LIN {X 0,Y 474.616,Z 278.985,A -85,B 0,C 180,E1 -7437.787,E2 -7437.787} C_VEL
LIN {X 0,Y 474.604,Z 278.989,A -85,B 0,C 180,E1 -7440.884,E2 -7440.884} C_VEL
LIN {X 0,Y 474.635,Z 278.982,A -85,B 0,C 180,E1 -7443.627,E2 -7443.627} C_VEL
LIN {X 0,Y 474.616,Z 278.99,A -85,B 0,C 180,E1 -7446.641,E2 -7446.641} C_VEL
LIN {X 0,Y 474.636,Z 278.981,A -85,B 0,C 180,E1 -7450.089,E2 -7450.089} C_VEL
LIN {X 0,Y 474.637,Z 278.985,A -85,B 0,C 180,E1 -7451.617,E2 -7451.617} C_VEL
LIN {X 0,Y 473.97,Z 279.072,A -85,B 0,C 180,E1 -7452.326,E2 -7452.326} C_VEL
LIN {X 0,Y 471.122,Z 279.425,A -85,B 0,C 180,E1 -7453.477,E2 -7453.477} C_VEL
LIN {X 0,Y 468.71,Z 279.726,A -85,B 0,C 180,E1 -7454.406,E2 -7454.406} C_VEL
LIN {X 0,Y 467.667,Z 279.855,A -85,B 0,C 180,E1 -7455.123,E2 -7455.123} C_VEL
LIN {X 0,Y 467.579,Z 279.864,A -85,B 0,C 180,E1 -7455.365,E2 -7455.365} C_VEL
LIN {X 0,Y 467.665,Z 279.853,A -85,B 0,C 180,E1 -7457.855,E2 -7457.855} C_VEL
LIN {X 0,Y 467.663,Z 279.853,A -85,B 0,C 180,E1 -7461.357,E2 -7461.357} C_VEL
LIN {X 0,Y 467.715,Z 279.848,A -85,B 0,C 180,E1 -7463.962,E2 -7463.962} C_VEL
LIN {X 0,Y 467.84,Z 279.834,A -85,B 0,C 180,E1 -7467.417,E2 -7467.417} C_VEL
LIN {X 0,Y 467.861,Z 279.836,A -85,B 0,C 180,E1 -7470,E2 -7470} C_VEL
LIN {X 0,Y 467.838,Z 279.841,A -85,B 0,C 180,E1 -7472.583,E2 -7472.583} C_VEL
LIN {X 0,Y 467.733,Z 280.061,A -85,B 0,C 180,E1 -7473.068,E2 -7473.068} C_VEL
LIN {X 0,Y 470.913,Z 294.475,A -85,B 0,C 180,E1 -7475.781,E2 -7475.781} C_VEL
LIN {X 0,Y 471.168,Z 295.669,A -85,B 0,C 180,E1 -7475.953,E2 -7475.953} C_VEL
LIN {X 0,Y 475.313,Z 312.707,A -85,B 0,C 180,E1 -7476.456,E2 -7476.456} C_VEL
LIN {X 0,Y 476.029,Z 316.068,A -85,B 0,C 180,E1 -7476.548,E2 -7476.548} C_VEL
LIN {X 0,Y 474.23,Z 459.892,A -85,B 0,C 180,E1 -7478.817,E2 -7478.817} C_VEL
LIN {X 0,Y 473.781,Z 475.482,A -85,B 0,C 180,E1 -7479.229,E2 -7479.229} C_VEL
LIN {X 0,Y 473.147,Z 491.137,A -85,B 0,C 180,E1 -7479.835,E2 -7479.835} C_VEL
LIN {X 0,Y 472.45,Z 505.523,A -85,B 0,C 180,E1 -7480.579,E2 -7480.579} C_VEL
LIN {X 0,Y 471.64,Z 519.544,A -85,B 0,C 180,E1 -7481.496,E2 -7481.496} C_VEL
LIN {X 0,Y 470.763,Z 533.282,A -85,B 0,C 180,E1 -7482.611,E2 -7482.611} C_VEL
LIN {X 0,Y 469.923,Z 545.755,A -85,B 0,C 180,E1 -7483.844,E2 -7483.844} C_VEL
LIN {X 0,Y 469.124,Z 557.142,A -85,B 0,C 180,E1 -7485.198,E2 -7485.198} C_VEL
LIN {X 0,Y 468.452,Z 566.781,A -85,B 0,C 180,E1 -7486.561,E2 -7486.561} C_VEL
LIN {X 0,Y 467.84,Z 576.198,A -85,B 0,C 180,E1 -7488.162,E2 -7488.162} C_VEL
LIN {X 0,Y 467.414,Z 584.01,A -85,B 0,C 180,E1 -7489.773,E2 -7489.773} C_VEL
LIN {X 0,Y 467.108,Z 589.576,A -85,B 0,C 180,E1 -7491.167,E2 -7491.167} C_VEL
LIN {X 0,Y 466.868,Z 595.614,A -85,B 0,C 180,E1 -7493.04,E2 -7493.04} C_VEL
LIN {X 0,Y 466.72,Z 600.136,A -85,B 0,C 180,E1 -7494.937,E2 -7494.937} C_VEL
LIN {X 0,Y 466.549,Z 603.229,A -85,B 0,C 180,E1 -7496.866,E2 -7496.866} C_VEL
LIN {X 0,Y 466.498,Z 604.884,A -85,B 0,C 180,E1 -7498.821,E2 -7498.821} C_VEL
LIN {X 0,Y 466.502,Z 605.166,A -85,B 0,C 180,E1 -7499.811,E2 -7499.811} C_VEL
LIN {X 0,Y 466.52,Z 605.07,A -85,B 0,C 180,E1 -7500.835,E2 -7500.835} C_VEL
LIN {X 0,Y 466.517,Z 603.726,A -85,B 0,C 180,E1 -7502.841,E2 -7502.841} C_VEL
LIN {X 0,Y 466.565,Z 602.133,A -85,B 0,C 180,E1 -7504.061,E2 -7504.061} C_VEL
LIN {X 0,Y 466.75,Z 599.272,A -85,B 0,C 180,E1 -7505.605,E2 -7505.605} C_VEL
LIN {X 0,Y 466.958,Z 594.255,A -85,B 0,C 180,E1 -7507.555,E2 -7507.555} C_VEL
LIN {X 0,Y 467.202,Z 588.729,A -85,B 0,C 180,E1 -7509.181,E2 -7509.181} C_VEL
LIN {X 0,Y 467.569,Z 581.995,A -85,B 0,C 180,E1 -7510.784,E2 -7510.784} C_VEL
LIN {X 0,Y 467.974,Z 574.714,A -85,B 0,C 180,E1 -7512.224,E2 -7512.224} C_VEL
LIN {X 0,Y 468.594,Z 565.162,A -85,B 0,C 180,E1 -7513.797,E2 -7513.797} C_VEL
LIN {X 0,Y 469.327,Z 554.381,A -85,B 0,C 180,E1 -7515.27,E2 -7515.27} C_VEL
LIN {X 0,Y 470.12,Z 543.077,A -85,B 0,C 180,E1 -7516.557,E2 -7516.557} C_VEL
LIN {X 0,Y 470.972,Z 530.595,A -85,B 0,C 180,E1 -7517.74,E2 -7517.74} C_VEL
LIN {X 0,Y 471.841,Z 517.282,A -85,B 0,C 180,E1 -7518.778,E2 -7518.778} C_VEL
LIN {X 0,Y 472.6,Z 503.49,A -85,B 0,C 180,E1 -7519.651,E2 -7519.651} C_VEL
LIN {X 0,Y 473.315,Z 489.065,A -85,B 0,C 180,E1 -7520.367,E2 -7520.367} C_VEL
LIN {X 0,Y 473.895,Z 474.26,A -85,B 0,C 180,E1 -7520.918,E2 -7520.918} C_VEL
LIN {X 0,Y 474.306,Z 459.493,A -85,B 0,C 180,E1 -7521.3,E2 -7521.3} C_VEL
LIN {X 0,Y 476.099,Z 315.733,A -85,B 0,C 180,E1 -7523.583,E2 -7523.583} C_VEL
LIN {X 0,Y 471.607,Z 297.104,A -85,B 0,C 180,E1 -7524.142,E2 -7524.142} C_VEL
LIN {X 0,Y 471.197,Z 295.69,A -85,B 0,C 180,E1 -7524.215,E2 -7524.215} C_VEL
LIN {X 0,Y 467.882,Z 281.102,A -85,B 0,C 180,E1 -7527.011,E2 -7527.011} C_VEL
LIN {X 0,Y 467.59,Z 279.867,A -85,B 0,C 180,E1 -7527.282,E2 -7527.282} C_VEL
LIN {X 0,Y 467.561,Z 279.87,A -85,B 0,C 180,E1 -7530.667,E2 -7530.667} C_VEL
LIN {X 0,Y 467.611,Z 279.862,A -85,B 0,C 180,E1 -7533.202,E2 -7533.202} C_VEL
LIN {X 0,Y 467.576,Z 279.867,A -85,B 0,C 180,E1 -7536.469,E2 -7536.469} C_VEL
LIN {X 0,Y 467.608,Z 279.863,A -85,B 0,C 180,E1 -7539.778,E2 -7539.778} C_VEL
LIN {X 0,Y 467.594,Z 279.864,A -85,B 0,C 180,E1 -7542.508,E2 -7542.508} C_VEL
LIN {X 0,Y 467.591,Z 279.867,A -85,B 0,C 180,E1 -7545.198,E2 -7545.198} C_VEL
LIN {X 0,Y 467.641,Z 279.857,A -85,B 0,C 180,E1 -7547.856,E2 -7547.856} C_VEL
LIN {X 0,Y 467.667,Z 279.856,A -85,B 0,C 180,E1 -7551.359,E2 -7551.359} C_VEL
LIN {X 0,Y 467.721,Z 279.843,A -85,B 0,C 180,E1 -7553.964,E2 -7553.964} C_VEL
LIN {X 0,Y 467.845,Z 279.833,A -85,B 0,C 180,E1 -7557.418,E2 -7557.418} C_VEL
LIN {X 0,Y 467.867,Z 279.827,A -85,B 0,C 180,E1 -7560.001,E2 -7560.001} C_VEL
LIN {X 0,Y 467.844,Z 279.831,A -85,B 0,C 180,E1 -7562.584,E2 -7562.584} C_VEL
LIN {X 0,Y 467.715,Z 279.846,A -85,B 0,C 180,E1 -7566.039,E2 -7566.039} C_VEL
LIN {X 0,Y 467.657,Z 279.856,A -85,B 0,C 180,E1 -7568.644,E2 -7568.644} C_VEL
LIN {X 0,Y 467.646,Z 279.855,A -85,B 0,C 180,E1 -7572.147,E2 -7572.147} C_VEL
LIN {X 0,Y 467.629,Z 279.857,A -85,B 0,C 180,E1 -7575.696,E2 -7575.696} C_VEL
LIN {X 0,Y 467.613,Z 279.858,A -85,B 0,C 180,E1 -7579.309,E2 -7579.309} C_VEL
LIN {X 0,Y 467.522,Z 279.873,A -85,B 0,C 180,E1 -7582.076,E2 -7582.076} C_VEL
LIN {X 0,Y 467.545,Z 279.869,A -85,B 0,C 180,E1 -7584.892,E2 -7584.892} C_VEL
LIN {X 0,Y 467.556,Z 279.867,A -85,B 0,C 180,E1 -7587.774,E2 -7587.774} C_VEL
LIN {X 0,Y 467.538,Z 279.866,A -85,B 0,C 180,E1 -7591.042,E2 -7591.042} C_VEL
LIN {X 0,Y 467.568,Z 279.867,A -85,B 0,C 180,E1 -7594.241,E2 -7594.241} C_VEL
LIN {X 0,Y 467.508,Z 279.87,A -85,B 0,C 180,E1 -7597.182,E2 -7597.182} C_VEL
LIN {X 0,Y 467.55,Z 279.873,A -85,B 0,C 180,E1 -7600.268,E2 -7600.268} C_VEL
LIN {X 0,Y 467.539,Z 279.871,A -85,B 0,C 180,E1 -7603.747,E2 -7603.747} C_VEL
LIN {X 0,Y 467.536,Z 279.875,A -85,B 0,C 180,E1 -7606.255,E2 -7606.255} C_VEL
LIN {X 0,Y 467.552,Z 279.871,A -85,B 0,C 180,E1 -7609.734,E2 -7609.734} C_VEL
LIN {X 0,Y 467.514,Z 279.868,A -85,B 0,C 180,E1 -7612.82,E2 -7612.82} C_VEL
LIN {X 0,Y 467.574,Z 279.866,A -85,B 0,C 180,E1 -7615.761,E2 -7615.761} C_VEL
LIN {X 0,Y 467.566,Z 279.868,A -85,B 0,C 180,E1 -7618.957,E2 -7618.957} C_VEL
LIN {X 0,Y 467.609,Z 279.998,A -85,B 0,C 180,E1 -7619.583,E2 -7619.583} C_VEL
LIN {X 0,Y 470.932,Z 293.674,A -85,B 0,C 180,E1 -7621.96,E2 -7621.96} C_VEL
LIN {X 0,Y 472.178,Z 299.765,A -85,B 0,C 180,E1 -7622.973,E2 -7622.973} C_VEL
LIN {X 0,Y 471.267,Z 317.413,A -85,B 0,C 180,E1 -7625.6,E2 -7625.6} C_VEL
LIN {X 0,Y 471.174,Z 319.057,A -85,B 0,C 180,E1 -7625.841,E2 -7625.841} C_VEL
LIN {X 0,Y 475.934,Z 344.308,A -85,B 0,C 180,E1 -7626.522,E2 -7626.522} C_VEL
LIN {X 0,Y 474.084,Z 485.77,A -85,B 0,C 180,E1 -7628.761,E2 -7628.761} C_VEL
LIN {X 0,Y 473.519,Z 501.577,A -85,B 0,C 180,E1 -7629.184,E2 -7629.184} C_VEL
LIN {X 0,Y 472.883,Z 517.077,A -85,B 0,C 180,E1 -7629.792,E2 -7629.792} C_VEL
LIN {X 0,Y 472.085,Z 531.609,A -85,B 0,C 180,E1 -7630.544,E2 -7630.544} C_VEL
LIN {X 0,Y 471.304,Z 544.953,A -85,B 0,C 180,E1 -7631.414,E2 -7631.414} C_VEL
LIN {X 0,Y 470.377,Z 558.527,A -85,B 0,C 180,E1 -7632.502,E2 -7632.502} C_VEL
LIN {X 0,Y 469.577,Z 570.878,A -85,B 0,C 180,E1 -7633.703,E2 -7633.703} C_VEL
LIN {X 0,Y 468.794,Z 582.148,A -85,B 0,C 180,E1 -7635.013,E2 -7635.013} C_VEL
LIN {X 0,Y 468.107,Z 593.098,A -85,B 0,C 180,E1 -7636.544,E2 -7636.544} C_VEL
LIN {X 0,Y 467.609,Z 602.208,A -85,B 0,C 180,E1 -7638.074,E2 -7638.074} C_VEL
LIN {X 0,Y 467.23,Z 609.763,A -85,B 0,C 180,E1 -7639.602,E2 -7639.602} C_VEL
LIN {X 0,Y 466.909,Z 616.818,A -85,B 0,C 180,E1 -7641.343,E2 -7641.343} C_VEL
LIN {X 0,Y 466.745,Z 622.369,A -85,B 0,C 180,E1 -7643.082,E2 -7643.082} C_VEL
LIN {X 0,Y 466.681,Z 626.569,A -85,B 0,C 180,E1 -7644.816,E2 -7644.816} C_VEL
LIN {X 0,Y 466.639,Z 629.514,A -85,B 0,C 180,E1 -7646.547,E2 -7646.547} C_VEL
LIN {X 0,Y 466.605,Z 631.274,A -85,B 0,C 180,E1 -7648.274,E2 -7648.274} C_VEL
LIN {X 0,Y 466.597,Z 631.882,A -85,B 0,C 180,E1 -7650,E2 -7650} C_VEL
LIN {X 0,Y 466.605,Z 631.287,A -85,B 0,C 180,E1 -7651.727,E2 -7651.727} C_VEL
LIN {X 0,Y 466.639,Z 629.54,A -85,B 0,C 180,E1 -7653.454,E2 -7653.454} C_VEL
LIN {X 0,Y 466.683,Z 626.612,A -85,B 0,C 180,E1 -7655.184,E2 -7655.184} C_VEL
LIN {X 0,Y 466.732,Z 622.433,A -85,B 0,C 180,E1 -7656.919,E2 -7656.919} C_VEL
LIN {X 0,Y 466.912,Z 616.895,A -85,B 0,C 180,E1 -7658.657,E2 -7658.657} C_VEL
LIN {X 0,Y 467.235,Z 609.848,A -85,B 0,C 180,E1 -7660.399,E2 -7660.399} C_VEL
LIN {X 0,Y 467.604,Z 602.308,A -85,B 0,C 180,E1 -7661.927,E2 -7661.927} C_VEL
LIN {X 0,Y 468.118,Z 593.215,A -85,B 0,C 180,E1 -7663.457,E2 -7663.457} C_VEL
LIN {X 0,Y 468.785,Z 582.268,A -85,B 0,C 180,E1 -7664.988,E2 -7664.988} C_VEL
LIN {X 0,Y 469.605,Z 571.008,A -85,B 0,C 180,E1 -7666.297,E2 -7666.297} C_VEL
LIN {X 0,Y 470.388,Z 558.653,A -85,B 0,C 180,E1 -7667.499,E2 -7667.499} C_VEL
LIN {X 0,Y 471.315,Z 545.044,A -85,B 0,C 180,E1 -7668.586,E2 -7668.586} C_VEL
LIN {X 0,Y 472.143,Z 531.671,A -85,B 0,C 180,E1 -7669.454,E2 -7669.454} C_VEL
LIN {X 0,Y 472.884,Z 516.979,A -85,B 0,C 180,E1 -7670.215,E2 -7670.215} C_VEL
LIN {X 0,Y 473.524,Z 501.724,A -85,B 0,C 180,E1 -7670.808,E2 -7670.808} C_VEL
LIN {X 0,Y 474.045,Z 486.623,A -85,B 0,C 180,E1 -7671.213,E2 -7671.213} C_VEL
LIN {X 0,Y 475.812,Z 343.392,A -85,B 0,C 180,E1 -7673.479,E2 -7673.479} C_VEL
LIN {X 0,Y 471.213,Z 319.394,A -85,B 0,C 180,E1 -7674.135,E2 -7674.135} C_VEL
LIN {X 0,Y 472.19,Z 301.71,A -85,B 0,C 180,E1 -7676.743,E2 -7676.743} C_VEL
LIN {X 0,Y 471.982,Z 298.347,A -85,B 0,C 180,E1 -7677.267,E2 -7677.267} C_VEL
LIN {X 0,Y 468.262,Z 282.598,A -85,B 0,C 180,E1 -7679.936,E2 -7679.936} C_VEL
LIN {X 0,Y 467.582,Z 279.858,A -85,B 0,C 180,E1 -7680.42,E2 -7680.42} C_VEL
LIN {X 0,Y 467.568,Z 279.87,A -85,B 0,C 180,E1 -7683.789,E2 -7683.789} C_VEL
LIN {X 0,Y 467.513,Z 279.876,A -85,B 0,C 180,E1 -7686.963,E2 -7686.963} C_VEL
LIN {X 0,Y 467.561,Z 279.871,A -85,B 0,C 180,E1 -7689.95,E2 -7689.95} C_VEL
LIN {X 0,Y 467.518,Z 279.871,A -85,B 0,C 180,E1 -7692.567,E2 -7692.567} C_VEL
LIN {X 0,Y 467.564,Z 279.866,A -85,B 0,C 180,E1 -7695.051,E2 -7695.051} C_VEL
LIN {X 0,Y 467.561,Z 279.869,A -85,B 0,C 180,E1 -7698.725,E2 -7698.725} C_VEL
LIN {X 0,Y 467.538,Z 279.874,A -85,B 0,C 180,E1 -7701.952,E2 -7701.952} C_VEL
LIN {X 0,Y 467.547,Z 279.864,A -85,B 0,C 180,E1 -7705.165,E2 -7705.165} C_VEL
LIN {X 0,Y 467.576,Z 279.866,A -85,B 0,C 180,E1 -7708.258,E2 -7708.258} C_VEL
LIN {X 0,Y 467.544,Z 279.868,A -85,B 0,C 180,E1 -7711.247,E2 -7711.247} C_VEL
LIN {X 0,Y 467.573,Z 279.867,A -85,B 0,C 180,E1 -7714.4,E2 -7714.4} C_VEL
LIN {X 0,Y 467.569,Z 279.864,A -85,B 0,C 180,E1 -7716.994,E2 -7716.994} C_VEL
LIN {X 0,Y 467.617,Z 279.864,A -85,B 0,C 180,E1 -7719.776,E2 -7719.776} C_VEL
LIN {X 0,Y 467.584,Z 279.864,A -85,B 0,C 180,E1 -7722.505,E2 -7722.505} C_VEL
LIN {X 0,Y 467.598,Z 279.86,A -85,B 0,C 180,E1 -7725.195,E2 -7725.195} C_VEL
LIN {X 0,Y 467.641,Z 279.846,A -85,B 0,C 180,E1 -7727.853,E2 -7727.853} C_VEL
LIN {X 0,Y 467.622,Z 279.86,A -85,B 0,C 180,E1 -7731.355,E2 -7731.355} C_VEL
LIN {X 0,Y 467.694,Z 279.847,A -85,B 0,C 180,E1 -7733.961,E2 -7733.961} C_VEL
LIN {X 0,Y 467.78,Z 279.827,A -85,B 0,C 180,E1 -7737.415,E2 -7737.415} C_VEL
LIN {X 0,Y 467.837,Z 279.832,A -85,B 0,C 180,E1 -7739.999,E2 -7739.999} C_VEL
LIN {X 0,Y 467.81,Z 279.833,A -85,B 0,C 180,E1 -7742.582,E2 -7742.582} C_VEL
LIN {X 0,Y 467.668,Z 279.835,A -85,B 0,C 180,E1 -7746.037,E2 -7746.037} C_VEL
LIN {X 0,Y 467.62,Z 279.85,A -85,B 0,C 180,E1 -7748.642,E2 -7748.642} C_VEL
LIN {X 0,Y 467.645,Z 279.854,A -85,B 0,C 180,E1 -7752.144,E2 -7752.144} C_VEL
LIN {X 0,Y 467.612,Z 279.845,A -85,B 0,C 180,E1 -7755.872,E2 -7755.872} C_VEL
LIN {X 0,Y 467.606,Z 279.857,A -85,B 0,C 180,E1 -7759.307,E2 -7759.307} C_VEL
LIN {X 0,Y 467.518,Z 279.87,A -85,B 0,C 180,E1 -7762.073,E2 -7762.073} C_VEL
LIN {X 0,Y 467.543,Z 279.866,A -85,B 0,C 180,E1 -7764.889,E2 -7764.889} C_VEL
LIN {X 0,Y 467.532,Z 279.859,A -85,B 0,C 180,E1 -7767.773,E2 -7767.773} C_VEL
LIN {X 0,Y 467.535,Z 279.871,A -85,B 0,C 180,E1 -7771.039,E2 -7771.039} C_VEL
LIN {X 0,Y 467.561,Z 279.861,A -85,B 0,C 180,E1 -7774.238,E2 -7774.238} C_VEL
LIN {X 0,Y 467.527,Z 279.861,A -85,B 0,C 180,E1 -7777.184,E2 -7777.184} C_VEL
LIN {X 0,Y 467.543,Z 279.866,A -85,B 0,C 180,E1 -7780.265,E2 -7780.265} C_VEL
LIN {X 0,Y 467.53,Z 279.863,A -85,B 0,C 180,E1 -7783.744,E2 -7783.744} C_VEL
LIN {X 0,Y 467.531,Z 279.86,A -85,B 0,C 180,E1 -7786.253,E2 -7786.253} C_VEL
LIN {X 0,Y 467.553,Z 279.867,A -85,B 0,C 180,E1 -7789.734,E2 -7789.734} C_VEL
LIN {X 0,Y 467.53,Z 279.866,A -85,B 0,C 180,E1 -7792.813,E2 -7792.813} C_VEL
LIN {X 0,Y 467.56,Z 279.866,A -85,B 0,C 180,E1 -7795.759,E2 -7795.759} C_VEL
LIN {X 0,Y 467.549,Z 279.865,A -85,B 0,C 180,E1 -7798.955,E2 -7798.955} C_VEL
LIN {X 0,Y 467.615,Z 279.861,A -85,B 0,C 180,E1 -7802.461,E2 -7802.461} C_VEL
LIN {X 0,Y 467.566,Z 279.865,A -85,B 0,C 180,E1 -7805.111,E2 -7805.111} C_VEL
LIN {X 0,Y 467.515,Z 279.872,A -85,B 0,C 180,E1 -7807.925,E2 -7807.925} C_VEL
LIN {X 0,Y 467.605,Z 279.863,A -85,B 0,C 180,E1 -7810.692,E2 -7810.692} C_VEL
LIN {X 0,Y 467.631,Z 279.855,A -85,B 0,C 180,E1 -7814.114,E2 -7814.114} C_VEL
LIN {X 0,Y 467.579,Z 279.864,A -85,B 0,C 180,E1 -7815.365,E2 -7815.365} C_VEL
LIN {X 0,Y 466.908,Z 279.949,A -85,B 0,C 180,E1 -7816.085,E2 -7816.085} C_VEL
LIN {X 0,Y 464.078,Z 280.301,A -85,B 0,C 180,E1 -7817.254,E2 -7817.254} C_VEL
LIN {X 0,Y 461.688,Z 280.6,A -85,B 0,C 180,E1 -7818.196,E2 -7818.196} C_VEL
LIN {X 0,Y 460.66,Z 280.727,A -85,B 0,C 180,E1 -7818.924,E2 -7818.924} C_VEL
LIN {X 0,Y 460.574,Z 280.735,A -85,B 0,C 180,E1 -7819.171,E2 -7819.171} C_VEL
LIN {X 0,Y 460.696,Z 280.724,A -85,B 0,C 180,E1 -7822.543,E2 -7822.543} C_VEL
LIN {X 0,Y 460.673,Z 280.73,A -85,B 0,C 180,E1 -7824.748,E2 -7824.748} C_VEL
LIN {X 0,Y 460.781,Z 280.713,A -85,B 0,C 180,E1 -7827.377,E2 -7827.377} C_VEL
LIN {X 0,Y 460.833,Z 280.712,A -85,B 0,C 180,E1 -7830,E2 -7830} C_VEL
LIN {X 0,Y 460.743,Z 280.769,A -85,B 0,C 180,E1 -7832.732,E2 -7832.732} C_VEL
LIN {X 0,Y 463.932,Z 295.469,A -85,B 0,C 180,E1 -7835.541,E2 -7835.541} C_VEL
LIN {X 0,Y 466.028,Z 301.756,A -85,B 0,C 180,E1 -7835.776,E2 -7835.776} C_VEL
LIN {X 0,Y 469.487,Z 316.93,A -85,B 0,C 180,E1 -7836.217,E2 -7836.217} C_VEL
LIN {X 0,Y 467.604,Z 459.938,A -85,B 0,C 180,E1 -7838.507,E2 -7838.507} C_VEL
LIN {X 0,Y 467.133,Z 475.592,A -85,B 0,C 180,E1 -7838.925,E2 -7838.925} C_VEL
LIN {X 0,Y 466.474,Z 491.271,A -85,B 0,C 180,E1 -7839.539,E2 -7839.539} C_VEL
LIN {X 0,Y 465.701,Z 506.169,A -85,B 0,C 180,E1 -7840.323,E2 -7840.323} C_VEL
LIN {X 0,Y 464.846,Z 520.117,A -85,B 0,C 180,E1 -7841.254,E2 -7841.254} C_VEL
LIN {X 0,Y 463.944,Z 533.476,A -85,B 0,C 180,E1 -7842.355,E2 -7842.355} C_VEL
LIN {X 0,Y 463.085,Z 545.752,A -85,B 0,C 180,E1 -7843.583,E2 -7843.583} C_VEL
LIN {X 0,Y 462.229,Z 557.341,A -85,B 0,C 180,E1 -7844.979,E2 -7844.979} C_VEL
LIN {X 0,Y 461.429,Z 567.948,A -85,B 0,C 180,E1 -7846.519,E2 -7846.519} C_VEL
LIN {X 0,Y 460.845,Z 576.409,A -85,B 0,C 180,E1 -7847.987,E2 -7847.987} C_VEL
LIN {X 0,Y 460.395,Z 584.217,A -85,B 0,C 180,E1 -7849.622,E2 -7849.622} C_VEL
LIN {X 0,Y 460.013,Z 590.619,A -85,B 0,C 180,E1 -7851.266,E2 -7851.266} C_VEL
LIN {X 0,Y 459.797,Z 595.821,A -85,B 0,C 180,E1 -7852.939,E2 -7852.939} C_VEL
LIN {X 0,Y 459.676,Z 599.363,A -85,B 0,C 180,E1 -7854.38,E2 -7854.38} C_VEL
LIN {X 0,Y 459.468,Z 602.807,A -85,B 0,C 180,E1 -7856.332,E2 -7856.332} C_VEL
LIN {X 0,Y 459.397,Z 604.814,A -85,B 0,C 180,E1 -7858.309,E2 -7858.309} C_VEL
LIN {X 0,Y 459.406,Z 605.276,A -85,B 0,C 180,E1 -7859.315,E2 -7859.315} C_VEL
LIN {X 0,Y 459.407,Z 605.075,A -85,B 0,C 180,E1 -7861.34,E2 -7861.34} C_VEL
LIN {X 0,Y 459.428,Z 604.077,A -85,B 0,C 180,E1 -7862.721,E2 -7862.721} C_VEL
LIN {X 0,Y 459.505,Z 601.783,A -85,B 0,C 180,E1 -7864.464,E2 -7864.464} C_VEL
LIN {X 0,Y 459.678,Z 599.098,A -85,B 0,C 180,E1 -7865.877,E2 -7865.877} C_VEL
LIN {X 0,Y 459.894,Z 594.438,A -85,B 0,C 180,E1 -7867.68,E2 -7867.68} C_VEL
LIN {X 0,Y 460.229,Z 587.885,A -85,B 0,C 180,E1 -7869.608,E2 -7869.608} C_VEL
LIN {X 0,Y 460.645,Z 580.519,A -85,B 0,C 180,E1 -7871.32,E2 -7871.32} C_VEL
LIN {X 0,Y 461.192,Z 571.688,A -85,B 0,C 180,E1 -7872.994,E2 -7872.994} C_VEL
LIN {X 0,Y 461.949,Z 561.623,A -85,B 0,C 180,E1 -7874.565,E2 -7874.565} C_VEL
LIN {X 0,Y 462.738,Z 550.444,A -85,B 0,C 180,E1 -7876.013,E2 -7876.013} C_VEL
LIN {X 0,Y 463.647,Z 539.019,A -85,B 0,C 180,E1 -7877.247,E2 -7877.247} C_VEL
LIN {X 0,Y 464.502,Z 526.637,A -85,B 0,C 180,E1 -7878.365,E2 -7878.365} C_VEL
LIN {X 0,Y 465.489,Z 512.252,A -85,B 0,C 180,E1 -7879.421,E2 -7879.421} C_VEL
LIN {X 0,Y 466.242,Z 498.321,A -85,B 0,C 180,E1 -7880.24,E2 -7880.24} C_VEL
LIN {X 0,Y 466.921,Z 484.068,A -85,B 0,C 180,E1 -7880.891,E2 -7880.891} C_VEL
LIN {X 0,Y 467.472,Z 469.118,A -85,B 0,C 180,E1 -7881.391,E2 -7881.391} C_VEL
LIN {X 0,Y 467.842,Z 453.452,A -85,B 0,C 180,E1 -7881.731,E2 -7881.731} C_VEL
LIN {X 0,Y 469.552,Z 316.696,A -85,B 0,C 180,E1 -7883.926,E2 -7883.926} C_VEL
LIN {X 0,Y 465.375,Z 299.332,A -85,B 0,C 180,E1 -7884.46,E2 -7884.46} C_VEL
LIN {X 0,Y 464.036,Z 295.934,A -85,B 0,C 180,E1 -7884.622,E2 -7884.622} C_VEL
LIN {X 0,Y 461.102,Z 282.991,A -85,B 0,C 180,E1 -7887.152,E2 -7887.152} C_VEL
LIN {X 0,Y 460.52,Z 280.75,A -85,B 0,C 180,E1 -7887.641,E2 -7887.641} C_VEL
LIN {X 0,Y 460.53,Z 280.747,A -85,B 0,C 180,E1 -7890.771,E2 -7890.771} C_VEL
LIN {X 0,Y 460.552,Z 280.744,A -85,B 0,C 180,E1 -7893.736,E2 -7893.736} C_VEL
LIN {X 0,Y 460.53,Z 280.746,A -85,B 0,C 180,E1 -7896.625,E2 -7896.625} C_VEL
LIN {X 0,Y 460.537,Z 280.748,A -85,B 0,C 180,E1 -7899.454,E2 -7899.454} C_VEL
LIN {X 0,Y 460.544,Z 280.742,A -85,B 0,C 180,E1 -7902.231,E2 -7902.231} C_VEL
LIN {X 0,Y 460.55,Z 280.745,A -85,B 0,C 180,E1 -7904.966,E2 -7904.966} C_VEL
LIN {X 0,Y 460.596,Z 280.735,A -85,B 0,C 180,E1 -7908.561,E2 -7908.561} C_VEL
LIN {X 0,Y 460.681,Z 280.722,A -85,B 0,C 180,E1 -7912.11,E2 -7912.11} C_VEL
LIN {X 0,Y 460.679,Z 280.725,A -85,B 0,C 180,E1 -7914.75,E2 -7914.75} C_VEL
LIN {X 0,Y 460.786,Z 280.713,A -85,B 0,C 180,E1 -7917.379,E2 -7917.379} C_VEL
LIN {X 0,Y 460.838,Z 280.702,A -85,B 0,C 180,E1 -7920.001,E2 -7920.001} C_VEL
LIN {X 0,Y 460.785,Z 280.711,A -85,B 0,C 180,E1 -7922.624,E2 -7922.624} C_VEL
LIN {X 0,Y 460.681,Z 280.723,A -85,B 0,C 180,E1 -7926.132,E2 -7926.132} C_VEL
LIN {X 0,Y 460.607,Z 280.736,A -85,B 0,C 180,E1 -7928.778,E2 -7928.778} C_VEL
LIN {X 0,Y 460.599,Z 280.735,A -85,B 0,C 180,E1 -7932.336,E2 -7932.336} C_VEL
LIN {X 0,Y 460.592,Z 280.735,A -85,B 0,C 180,E1 -7935.999,E2 -7935.999} C_VEL
LIN {X 0,Y 460.559,Z 280.736,A -85,B 0,C 180,E1 -7939.617,E2 -7939.617} C_VEL
LIN {X 0,Y 460.499,Z 280.75,A -85,B 0,C 180,E1 -7942.43,E2 -7942.43} C_VEL
LIN {X 0,Y 460.515,Z 280.743,A -85,B 0,C 180,E1 -7945.792,E2 -7945.792} C_VEL
LIN {X 0,Y 460.511,Z 280.748,A -85,B 0,C 180,E1 -7948.237,E2 -7948.237} C_VEL
LIN {X 0,Y 460.514,Z 280.74,A -85,B 0,C 180,E1 -7951.284,E2 -7951.284} C_VEL
LIN {X 0,Y 460.512,Z 280.746,A -85,B 0,C 180,E1 -7954.504,E2 -7954.504} C_VEL
LIN {X 0,Y 460.476,Z 280.748,A -85,B 0,C 180,E1 -7957.627,E2 -7957.627} C_VEL
LIN {X 0,Y 460.508,Z 280.743,A -85,B 0,C 180,E1 -7961.015,E2 -7961.015} C_VEL
LIN {X 0,Y 460.505,Z 280.747,A -85,B 0,C 180,E1 -7964.591,E2 -7964.591} C_VEL
LIN {X 0,Y 460.469,Z 280.753,A -85,B 0,C 180,E1 -7967.814,E2 -7967.814} C_VEL
LIN {X 0,Y 460.506,Z 280.751,A -85,B 0,C 180,E1 -7970.136,E2 -7970.136} C_VEL
LIN {X 0,Y 460.458,Z 280.749,A -85,B 0,C 180,E1 -7973.47,E2 -7973.47} C_VEL
LIN {X 0,Y 460.518,Z 280.746,A -85,B 0,C 180,E1 -7976.676,E2 -7976.676} C_VEL
LIN {X 0,Y 460.546,Z 280.872,A -85,B 0,C 180,E1 -7979.225,E2 -7979.225} C_VEL
LIN {X 0,Y 463.742,Z 293.76,A -85,B 0,C 180,E1 -7981.522,E2 -7981.522} C_VEL
LIN {X 0,Y 465.371,Z 301.369,A -85,B 0,C 180,E1 -7982.819,E2 -7982.819} C_VEL
LIN {X 0,Y 464.458,Z 318.173,A -85,B 0,C 180,E1 -7985.356,E2 -7985.356} C_VEL
LIN {X 0,Y 464.421,Z 318.815,A -85,B 0,C 180,E1 -7985.453,E2 -7985.453} C_VEL
LIN {X 0,Y 469.409,Z 344.559,A -85,B 0,C 180,E1 -7986.176,E2 -7986.176} C_VEL
LIN {X 0,Y 467.484,Z 485.635,A -85,B 0,C 180,E1 -7988.446,E2 -7988.446} C_VEL
LIN {X 0,Y 466.882,Z 501.556,A -85,B 0,C 180,E1 -7988.88,E2 -7988.88} C_VEL
LIN {X 0,Y 466.183,Z 517.24,A -85,B 0,C 180,E1 -7989.507,E2 -7989.507} C_VEL
LIN {X 0,Y 465.368,Z 531.398,A -85,B 0,C 180,E1 -7990.251,E2 -7990.251} C_VEL
LIN {X 0,Y 464.535,Z 544.736,A -85,B 0,C 180,E1 -7991.133,E2 -7991.133} C_VEL
LIN {X 0,Y 463.548,Z 558.308,A -85,B 0,C 180,E1 -7992.235,E2 -7992.235} C_VEL
LIN {X 0,Y 462.71,Z 570.662,A -85,B 0,C 180,E1 -7993.454,E2 -7993.454} C_VEL
LIN {X 0,Y 461.85,Z 581.931,A -85,B 0,C 180,E1 -7994.783,E2 -7994.783} C_VEL
LIN {X 0,Y 461.124,Z 592.88,A -85,B 0,C 180,E1 -7996.336,E2 -7996.336} C_VEL
LIN {X 0,Y 460.588,Z 601.99,A -85,B 0,C 180,E1 -7997.89,E2 -7997.89} C_VEL
LIN {X 0,Y 460.209,Z 609.549,A -85,B 0,C 180,E1 -7999.441,E2 -7999.441} C_VEL
LIN {X 0,Y 459.851,Z 616.608,A -85,B 0,C 180,E1 -8001.209,E2 -8001.209} C_VEL
LIN {X 0,Y 459.666,Z 622.161,A -85,B 0,C 180,E1 -8002.975,E2 -8002.975} C_VEL
LIN {X 0,Y 459.588,Z 626.362,A -85,B 0,C 180,E1 -8004.736,E2 -8004.736} C_VEL
LIN {X 0,Y 459.536,Z 629.309,A -85,B 0,C 180,E1 -8006.493,E2 -8006.493} C_VEL
LIN {X 0,Y 459.518,Z 631.07,A -85,B 0,C 180,E1 -8008.248,E2 -8008.248} C_VEL
LIN {X 0,Y 459.528,Z 631.68,A -85,B 0,C 180,E1 -8010,E2 -8010} C_VEL
LIN {X 0,Y 459.518,Z 631.085,A -85,B 0,C 180,E1 -8011.753,E2 -8011.753} C_VEL
LIN {X 0,Y 459.536,Z 629.335,A -85,B 0,C 180,E1 -8013.508,E2 -8013.508} C_VEL
LIN {X 0,Y 459.593,Z 626.405,A -85,B 0,C 180,E1 -8015.265,E2 -8015.265} C_VEL
LIN {X 0,Y 459.655,Z 622.223,A -85,B 0,C 180,E1 -8017.026,E2 -8017.026} C_VEL
LIN {X 0,Y 459.856,Z 616.679,A -85,B 0,C 180,E1 -8018.791,E2 -8018.791} C_VEL
LIN {X 0,Y 460.22,Z 609.625,A -85,B 0,C 180,E1 -8020.559,E2 -8020.559} C_VEL
LIN {X 0,Y 460.579,Z 602.077,A -85,B 0,C 180,E1 -8022.111,E2 -8022.111} C_VEL
LIN {X 0,Y 461.133,Z 592.978,A -85,B 0,C 180,E1 -8023.664,E2 -8023.664} C_VEL
LIN {X 0,Y 461.847,Z 582.019,A -85,B 0,C 180,E1 -8025.218,E2 -8025.218} C_VEL
LIN {X 0,Y 462.733,Z 570.748,A -85,B 0,C 180,E1 -8026.545,E2 -8026.545} C_VEL
LIN {X 0,Y 463.567,Z 558.374,A -85,B 0,C 180,E1 -8027.765,E2 -8027.765} C_VEL
LIN {X 0,Y 464.551,Z 544.738,A -85,B 0,C 180,E1 -8028.867,E2 -8028.867} C_VEL
LIN {X 0,Y 465.42,Z 531.341,A -85,B 0,C 180,E1 -8029.747,E2 -8029.747} C_VEL
LIN {X 0,Y 466.155,Z 517.045,A -85,B 0,C 180,E1 -8030.497,E2 -8030.497} C_VEL
LIN {X 0,Y 466.841,Z 501.245,A -85,B 0,C 180,E1 -8031.122,E2 -8031.122} C_VEL
LIN {X 0,Y 467.428,Z 486.079,A -85,B 0,C 180,E1 -8031.528,E2 -8031.528} C_VEL
LIN {X 0,Y 469.276,Z 344.848,A -85,B 0,C 180,E1 -8033.792,E2 -8033.792} C_VEL
LIN {X 0,Y 464.43,Z 319.251,A -85,B 0,C 180,E1 -8034.496,E2 -8034.496} C_VEL
LIN {X 0,Y 465.399,Z 302.518,A -85,B 0,C 180,E1 -8037.005,E2 -8037.005} C_VEL
LIN {X 0,Y 464.355,Z 296.62,A -85,B 0,C 180,E1 -8037.981,E2 -8037.981} C_VEL
LIN {X 0,Y 460.942,Z 282.34,A -85,B 0,C 180,E1 -8040.461,E2 -8040.461} C_VEL
LIN {X 0,Y 460.549,Z 280.736,A -85,B 0,C 180,E1 -8040.776,E2 -8040.776} C_VEL
LIN {X 0,Y 460.518,Z 280.747,A -85,B 0,C 180,E1 -8043.325,E2 -8043.325} C_VEL
LIN {X 0,Y 460.466,Z 280.757,A -85,B 0,C 180,E1 -8046.53,E2 -8046.53} C_VEL
LIN {X 0,Y 460.51,Z 280.75,A -85,B 0,C 180,E1 -8049.864,E2 -8049.864} C_VEL
LIN {X 0,Y 460.461,Z 280.748,A -85,B 0,C 180,E1 -8052.892,E2 -8052.892} C_VEL
LIN {X 0,Y 460.503,Z 280.749,A -85,B 0,C 180,E1 -8055.831,E2 -8055.831} C_VEL
LIN {X 0,Y 460.515,Z 280.746,A -85,B 0,C 180,E1 -8058.986,E2 -8058.986} C_VEL
LIN {X 0,Y 460.481,Z 280.753,A -85,B 0,C 180,E1 -8062.374,E2 -8062.374} C_VEL
LIN {X 0,Y 460.531,Z 280.739,A -85,B 0,C 180,E1 -8065.621,E2 -8065.621} C_VEL
LIN {X 0,Y 460.519,Z 280.742,A -85,B 0,C 180,E1 -8068.742,E2 -8068.742} C_VEL
LIN {X 0,Y 460.506,Z 280.751,A -85,B 0,C 180,E1 -8071.763,E2 -8071.763} C_VEL
LIN {X 0,Y 460.516,Z 280.744,A -85,B 0,C 180,E1 -8074.702,E2 -8074.702} C_VEL
LIN {X 0,Y 460.504,Z 280.749,A -85,B 0,C 180,E1 -8077.57,E2 -8077.57} C_VEL
LIN {X 0,Y 460.562,Z 280.737,A -85,B 0,C 180,E1 -8080.383,E2 -8080.383} C_VEL
LIN {X 0,Y 460.575,Z 280.737,A -85,B 0,C 180,E1 -8084.011,E2 -8084.011} C_VEL
LIN {X 0,Y 460.597,Z 280.721,A -85,B 0,C 180,E1 -8087.664,E2 -8087.664} C_VEL
LIN {X 0,Y 460.577,Z 280.736,A -85,B 0,C 180,E1 -8091.222,E2 -8091.222} C_VEL
LIN {X 0,Y 460.661,Z 280.724,A -85,B 0,C 180,E1 -8093.868,E2 -8093.868} C_VEL
LIN {X 0,Y 460.727,Z 280.704,A -85,B 0,C 180,E1 -8097.376,E2 -8097.376} C_VEL
LIN {X 0,Y 460.786,Z 280.71,A -85,B 0,C 180,E1 -8099.999,E2 -8099.999} C_VEL
LIN {X 0,Y 460.755,Z 280.712,A -85,B 0,C 180,E1 -8102.621,E2 -8102.621} C_VEL
LIN {X 0,Y 460.633,Z 280.71,A -85,B 0,C 180,E1 -8106.129,E2 -8106.129} C_VEL
LIN {X 0,Y 460.575,Z 280.727,A -85,B 0,C 180,E1 -8108.776,E2 -8108.776} C_VEL
LIN {X 0,Y 460.599,Z 280.732,A -85,B 0,C 180,E1 -8112.333,E2 -8112.333} C_VEL
LIN {X 0,Y 460.568,Z 280.721,A -85,B 0,C 180,E1 -8115.986,E2 -8115.986} C_VEL
LIN {X 0,Y 460.553,Z 280.739,A -85,B 0,C 180,E1 -8119.614,E2 -8119.614} C_VEL
LIN {X 0,Y 460.494,Z 280.745,A -85,B 0,C 180,E1 -8122.427,E2 -8122.427} C_VEL
LIN {X 0,Y 460.519,Z 280.73,A -85,B 0,C 180,E1 -8125.791,E2 -8125.791} C_VEL
LIN {X 0,Y 460.506,Z 280.741,A -85,B 0,C 180,E1 -8129.231,E2 -8129.231} C_VEL
LIN {X 0,Y 460.511,Z 280.743,A -85,B 0,C 180,E1 -8132.284,E2 -8132.284} C_VEL
LIN {X 0,Y 460.491,Z 280.736,A -85,B 0,C 180,E1 -8135.445,E2 -8135.445} C_VEL
LIN {X 0,Y 460.489,Z 280.743,A -85,B 0,C 180,E1 -8138.89,E2 -8138.89} C_VEL
LIN {X 0,Y 460.493,Z 280.747,A -85,B 0,C 180,E1 -8141.598,E2 -8141.598} C_VEL
LIN {X 0,Y 460.495,Z 280.741,A -85,B 0,C 180,E1 -8144.588,E2 -8144.588} C_VEL
LIN {X 0,Y 460.487,Z 280.746,A -85,B 0,C 180,E1 -8147.815,E2 -8147.815} C_VEL
LIN {X 0,Y 460.522,Z 280.743,A -85,B 0,C 180,E1 -8151.102,E2 -8151.102} C_VEL
LIN {X 0,Y 460.491,Z 280.743,A -85,B 0,C 180,E1 -8154.553,E2 -8154.553} C_VEL
LIN {X 0,Y 460.512,Z 280.742,A -85,B 0,C 180,E1 -8157.714,E2 -8157.714} C_VEL
LIN {X 0,Y 460.52,Z 280.741,A -85,B 0,C 180,E1 -8160.768,E2 -8160.768} C_VEL
LIN {X 0,Y 460.538,Z 280.738,A -85,B 0,C 180,E1 -8163.733,E2 -8163.733} C_VEL
LIN {X 0,Y 460.526,Z 280.745,A -85,B 0,C 180,E1 -8166.623,E2 -8166.623} C_VEL
LIN {X 0,Y 460.532,Z 280.738,A -85,B 0,C 180,E1 -8169.452,E2 -8169.452} C_VEL
LIN {X 0,Y 460.539,Z 280.743,A -85,B 0,C 180,E1 -8172.229,E2 -8172.229} C_VEL
LIN {X 0,Y 460.546,Z 280.744,A -85,B 0,C 180,E1 -8174.964,E2 -8174.964} C_VEL
LIN {X 0,Y 460.612,Z 280.731,A -85,B 0,C 180,E1 -8177.666,E2 -8177.666} C_VEL
LIN {X 0,Y 460.574,Z 280.735,A -85,B 0,C 180,E1 -8179.171,E2 -8179.171} C_VEL
LIN {X 0,Y 459.909,Z 280.817,A -85,B 0,C 180,E1 -8179.901,E2 -8179.901} C_VEL
LIN {X 0,Y 457.084,Z 281.174,A -85,B 0,C 180,E1 -8181.087,E2 -8181.087} C_VEL
LIN {X 0,Y 454.703,Z 281.475,A -85,B 0,C 180,E1 -8182.044,E2 -8182.044} C_VEL
LIN {X 0,Y 453.688,Z 281.6,A -85,B 0,C 180,E1 -8182.782,E2 -8182.782} C_VEL
LIN {X 0,Y 453.609,Z 281.607,A -85,B 0,C 180,E1 -8183.032,E2 -8183.032} C_VEL
LIN {X 0,Y 453.647,Z 281.604,A -85,B 0,C 180,E1 -8184.666,E2 -8184.666} C_VEL
LIN {X 0,Y 453.725,Z 281.593,A -85,B 0,C 180,E1 -8187.336,E2 -8187.336} C_VEL
LIN {X 0,Y 453.804,Z 281.588,A -85,B 0,C 180,E1 -8190,E2 -8190} C_VEL
LIN {X 0,Y 453.734,Z 281.801,A -85,B 0,C 180,E1 -8192.441,E2 -8192.441} C_VEL
LIN {X 0,Y 456.812,Z 295.848,A -85,B 0,C 180,E1 -8195.158,E2 -8195.158} C_VEL
LIN {X 0,Y 459.689,Z 303.581,A -85,B 0,C 180,E1 -8195.455,E2 -8195.455} C_VEL
LIN {X 0,Y 462.926,Z 317.965,A -85,B 0,C 180,E1 -8195.881,E2 -8195.881} C_VEL
LIN {X 0,Y 460.935,Z 461.327,A -85,B 0,C 180,E1 -8198.218,E2 -8198.218} C_VEL
LIN {X 0,Y 460.425,Z 477.303,A -85,B 0,C 180,E1 -8198.669,E2 -8198.669} C_VEL
LIN {X 0,Y 459.728,Z 492.569,A -85,B 0,C 180,E1 -8199.292,E2 -8199.292} C_VEL
LIN {X 0,Y 459.02,Z 506.292,A -85,B 0,C 180,E1 -8200.029,E2 -8200.029} C_VEL
LIN {X 0,Y 458.117,Z 520.021,A -85,B 0,C 180,E1 -8200.953,E2 -8200.953} C_VEL
LIN {X 0,Y 457.172,Z 533.639,A -85,B 0,C 180,E1 -8202.09,E2 -8202.09} C_VEL
LIN {X 0,Y 456.224,Z 546.136,A -85,B 0,C 180,E1 -8203.359,E2 -8203.359} C_VEL
LIN {X 0,Y 455.325,Z 557.537,A -85,B 0,C 180,E1 -8204.754,E2 -8204.754} C_VEL
LIN {X 0,Y 454.574,Z 567.182,A -85,B 0,C 180,E1 -8206.157,E2 -8206.157} C_VEL
LIN {X 0,Y 453.864,Z 576.609,A -85,B 0,C 180,E1 -8207.807,E2 -8207.807} C_VEL
LIN {X 0,Y 453.369,Z 584.422,A -85,B 0,C 180,E1 -8209.467,E2 -8209.467} C_VEL
LIN {X 0,Y 453.029,Z 589.986,A -85,B 0,C 180,E1 -8210.903,E2 -8210.903} C_VEL
LIN {X 0,Y 452.722,Z 596.028,A -85,B 0,C 180,E1 -8212.835,E2 -8212.835} C_VEL
LIN {X 0,Y 452.597,Z 599.567,A -85,B 0,C 180,E1 -8214.298,E2 -8214.298} C_VEL
LIN {X 0,Y 452.424,Z 602.276,A -85,B 0,C 180,E1 -8215.781,E2 -8215.781} C_VEL
LIN {X 0,Y 452.305,Z 604.647,A -85,B 0,C 180,E1 -8217.783,E2 -8217.783} C_VEL
LIN {X 0,Y 452.291,Z 605.574,A -85,B 0,C 180,E1 -8219.816,E2 -8219.816} C_VEL
LIN {X 0,Y 452.315,Z 605.317,A -85,B 0,C 180,E1 -8221.291,E2 -8221.291} C_VEL
LIN {X 0,Y 452.332,Z 604.103,A -85,B 0,C 180,E1 -8222.968,E2 -8222.968} C_VEL
LIN {X 0,Y 452.421,Z 601.906,A -85,B 0,C 180,E1 -8224.586,E2 -8224.586} C_VEL
LIN {X 0,Y 452.618,Z 598.866,A -85,B 0,C 180,E1 -8226.159,E2 -8226.159} C_VEL
LIN {X 0,Y 452.869,Z 594.098,A -85,B 0,C 180,E1 -8227.984,E2 -8227.984} C_VEL
LIN {X 0,Y 453.193,Z 588.104,A -85,B 0,C 180,E1 -8229.756,E2 -8229.756} C_VEL
LIN {X 0,Y 453.644,Z 580.841,A -85,B 0,C 180,E1 -8231.474,E2 -8231.474} C_VEL
LIN {X 0,Y 454.213,Z 572.231,A -85,B 0,C 180,E1 -8233.139,E2 -8233.139} C_VEL
LIN {X 0,Y 455.023,Z 562.27,A -85,B 0,C 180,E1 -8234.729,E2 -8234.729} C_VEL
LIN {X 0,Y 455.839,Z 551.197,A -85,B 0,C 180,E1 -8236.198,E2 -8236.198} C_VEL
LIN {X 0,Y 456.768,Z 540.385,A -85,B 0,C 180,E1 -8237.393,E2 -8237.393} C_VEL
LIN {X 0,Y 457.713,Z 527.45,A -85,B 0,C 180,E1 -8238.595,E2 -8238.595} C_VEL
LIN {X 0,Y 458.726,Z 513.382,A -85,B 0,C 180,E1 -8239.657,E2 -8239.657} C_VEL
LIN {X 0,Y 459.544,Z 499.573,A -85,B 0,C 180,E1 -8240.492,E2 -8240.492} C_VEL
LIN {X 0,Y 460.313,Z 484.301,A -85,B 0,C 180,E1 -8241.207,E2 -8241.207} C_VEL
LIN {X 0,Y 460.895,Z 469.112,A -85,B 0,C 180,E1 -8241.721,E2 -8241.721} C_VEL
LIN {X 0,Y 461.293,Z 453.001,A -85,B 0,C 180,E1 -8242.071,E2 -8242.071} C_VEL
LIN {X 0,Y 463.141,Z 318.718,A -85,B 0,C 180,E1 -8244.254,E2 -8244.254} C_VEL
LIN {X 0,Y 460.801,Z 307.69,A -85,B 0,C 180,E1 -8244.583,E2 -8244.583} C_VEL
LIN {X 0,Y 459.053,Z 301.506,A -85,B 0,C 180,E1 -8244.795,E2 -8244.795} C_VEL
LIN {X 0,Y 456.907,Z 296.199,A -85,B 0,C 180,E1 -8245.041,E2 -8245.041} C_VEL
LIN {X 0,Y 454.056,Z 284.082,A -85,B 0,C 180,E1 -8247.464,E2 -8247.464} C_VEL
LIN {X 0,Y 453.475,Z 281.625,A -85,B 0,C 180,E1 -8248.008,E2 -8248.008} C_VEL
LIN {X 0,Y 453.499,Z 281.621,A -85,B 0,C 180,E1 -8251.29,E2 -8251.29} C_VEL
LIN {X 0,Y 453.509,Z 281.619,A -85,B 0,C 180,E1 -8254.286,E2 -8254.286} C_VEL
LIN {X 0,Y 453.463,Z 281.627,A -85,B 0,C 180,E1 -8257.205,E2 -8257.205} C_VEL
LIN {X 0,Y 453.49,Z 281.62,A -85,B 0,C 180,E1 -8260.067,E2 -8260.067} C_VEL
LIN {X 0,Y 453.492,Z 281.624,A -85,B 0,C 180,E1 -8262.877,E2 -8262.877} C_VEL
LIN {X 0,Y 453.498,Z 281.621,A -85,B 0,C 180,E1 -8265.645,E2 -8265.645} C_VEL
LIN {X 0,Y 453.545,Z 281.613,A -85,B 0,C 180,E1 -8268.38,E2 -8268.38} C_VEL
LIN {X 0,Y 453.638,Z 281.6,A -85,B 0,C 180,E1 -8271.987,E2 -8271.987} C_VEL
LIN {X 0,Y 453.652,Z 281.599,A -85,B 0,C 180,E1 -8274.668,E2 -8274.668} C_VEL
LIN {X 0,Y 453.731,Z 281.592,A -85,B 0,C 180,E1 -8277.338,E2 -8277.338} C_VEL
LIN {X 0,Y 453.809,Z 281.578,A -85,B 0,C 180,E1 -8280.001,E2 -8280.001} C_VEL
LIN {X 0,Y 453.729,Z 281.59,A -85,B 0,C 180,E1 -8282.665,E2 -8282.665} C_VEL
LIN {X 0,Y 453.649,Z 281.599,A -85,B 0,C 180,E1 -8286.227,E2 -8286.227} C_VEL
LIN {X 0,Y 453.573,Z 281.614,A -85,B 0,C 180,E1 -8288.915,E2 -8288.915} C_VEL
LIN {X 0,Y 453.554,Z 281.615,A -85,B 0,C 180,E1 -8292.53,E2 -8292.53} C_VEL
LIN {X 0,Y 453.536,Z 281.615,A -85,B 0,C 180,E1 -8296.197,E2 -8296.197} C_VEL
LIN {X 0,Y 453.508,Z 281.617,A -85,B 0,C 180,E1 -8299.041,E2 -8299.041} C_VEL
LIN {X 0,Y 453.467,Z 281.622,A -85,B 0,C 180,E1 -8301.838,E2 -8301.838} C_VEL
LIN {X 0,Y 453.456,Z 281.626,A -85,B 0,C 180,E1 -8304.739,E2 -8304.739} C_VEL
LIN {X 0,Y 453.47,Z 281.623,A -85,B 0,C 180,E1 -8307.948,E2 -8307.948} C_VEL
LIN {X 0,Y 453.45,Z 281.623,A -85,B 0,C 180,E1 -8310.763,E2 -8310.763} C_VEL
LIN {X 0,Y 453.458,Z 281.624,A -85,B 0,C 180,E1 -8313.915,E2 -8313.915} C_VEL
LIN {X 0,Y 453.428,Z 281.624,A -85,B 0,C 180,E1 -8317.193,E2 -8317.193} C_VEL
LIN {X 0,Y 453.465,Z 281.623,A -85,B 0,C 180,E1 -8320.613,E2 -8320.613} C_VEL
LIN {X 0,Y 453.475,Z 281.624,A -85,B 0,C 180,E1 -8324.529,E2 -8324.529} C_VEL
LIN {X 0,Y 453.431,Z 281.631,A -85,B 0,C 180,E1 -8328.073,E2 -8328.073} C_VEL
LIN {X 0,Y 453.435,Z 281.628,A -85,B 0,C 180,E1 -8330.804,E2 -8330.804} C_VEL
LIN {X 0,Y 453.441,Z 281.628,A -85,B 0,C 180,E1 -8333.917,E2 -8333.917} C_VEL
LIN {X 0,Y 453.477,Z 281.623,A -85,B 0,C 180,E1 -8337.152,E2 -8337.152} C_VEL
LIN {X 0,Y 453.497,Z 281.689,A -85,B 0,C 180,E1 -8338.844,E2 -8338.844} C_VEL
LIN {X 0,Y 456.829,Z 295.024,A -85,B 0,C 180,E1 -8341.272,E2 -8341.272} C_VEL
LIN {X 0,Y 458.578,Z 303.452,A -85,B 0,C 180,E1 -8342.735,E2 -8342.735} C_VEL
LIN {X 0,Y 457.678,Z 318.599,A -85,B 0,C 180,E1 -8345.057,E2 -8345.057} C_VEL
LIN {X 0,Y 462.925,Z 345.768,A -85,B 0,C 180,E1 -8345.838,E2 -8345.838} C_VEL
LIN {X 0,Y 460.892,Z 485.554,A -85,B 0,C 180,E1 -8348.122,E2 -8348.122} C_VEL
LIN {X 0,Y 460.268,Z 501.414,A -85,B 0,C 180,E1 -8348.562,E2 -8348.562} C_VEL
LIN {X 0,Y 459.559,Z 516.134,A -85,B 0,C 180,E1 -8349.15,E2 -8349.15} C_VEL
LIN {X 0,Y 458.653,Z 531.205,A -85,B 0,C 180,E1 -8349.95,E2 -8349.95} C_VEL
LIN {X 0,Y 457.761,Z 544.539,A -85,B 0,C 180,E1 -8350.843,E2 -8350.843} C_VEL
LIN {X 0,Y 456.738,Z 558.106,A -85,B 0,C 180,E1 -8351.961,E2 -8351.961} C_VEL
LIN {X 0,Y 455.841,Z 570.454,A -85,B 0,C 180,E1 -8353.198,E2 -8353.198} C_VEL
LIN {X 0,Y 454.933,Z 581.719,A -85,B 0,C 180,E1 -8354.545,E2 -8354.545} C_VEL
LIN {X 0,Y 454.147,Z 592.669,A -85,B 0,C 180,E1 -8356.122,E2 -8356.122} C_VEL
LIN {X 0,Y 453.556,Z 601.493,A -85,B 0,C 180,E1 -8357.645,E2 -8357.645} C_VEL
LIN {X 0,Y 453.174,Z 609.341,A -85,B 0,C 180,E1 -8359.275,E2 -8359.275} C_VEL
LIN {X 0,Y 452.781,Z 616.399,A -85,B 0,C 180,E1 -8361.071,E2 -8361.071} C_VEL
LIN {X 0,Y 452.587,Z 621.954,A -85,B 0,C 180,E1 -8362.864,E2 -8362.864} C_VEL
LIN {X 0,Y 452.498,Z 626.157,A -85,B 0,C 180,E1 -8364.653,E2 -8364.653} C_VEL
LIN {X 0,Y 452.433,Z 629.105,A -85,B 0,C 180,E1 -8366.438,E2 -8366.438} C_VEL
LIN {X 0,Y 452.434,Z 630.868,A -85,B 0,C 180,E1 -8368.22,E2 -8368.22} C_VEL
LIN {X 0,Y 452.433,Z 631.477,A -85,B 0,C 180,E1 -8370,E2 -8370} C_VEL
LIN {X 0,Y 452.435,Z 630.881,A -85,B 0,C 180,E1 -8371.781,E2 -8371.781} C_VEL
LIN {X 0,Y 452.433,Z 629.129,A -85,B 0,C 180,E1 -8373.563,E2 -8373.563} C_VEL
LIN {X 0,Y 452.506,Z 626.196,A -85,B 0,C 180,E1 -8375.347,E2 -8375.347} C_VEL
LIN {X 0,Y 452.578,Z 622.009,A -85,B 0,C 180,E1 -8377.137,E2 -8377.137} C_VEL
LIN {X 0,Y 452.788,Z 616.46,A -85,B 0,C 180,E1 -8378.929,E2 -8378.929} C_VEL
LIN {X 0,Y 453.165,Z 609.399,A -85,B 0,C 180,E1 -8380.726,E2 -8380.726} C_VEL
LIN {X 0,Y 453.553,Z 601.564,A -85,B 0,C 180,E1 -8382.354,E2 -8382.354} C_VEL
LIN {X 0,Y 454.154,Z 592.733,A -85,B 0,C 180,E1 -8383.878,E2 -8383.878} C_VEL
LIN {X 0,Y 454.902,Z 581.755,A -85,B 0,C 180,E1 -8385.456,E2 -8385.456} C_VEL
LIN {X 0,Y 455.848,Z 570.471,A -85,B 0,C 180,E1 -8386.803,E2 -8386.803} C_VEL
LIN {X 0,Y 456.748,Z 558.082,A -85,B 0,C 180,E1 -8388.039,E2 -8388.039} C_VEL
LIN {X 0,Y 457.762,Z 544.419,A -85,B 0,C 180,E1 -8389.158,E2 -8389.158} C_VEL
LIN {X 0,Y 458.688,Z 531.002,A -85,B 0,C 180,E1 -8390.049,E2 -8390.049} C_VEL
LIN {X 0,Y 459.464,Z 517.081,A -85,B 0,C 180,E1 -8390.788,E2 -8390.788} C_VEL
LIN {X 0,Y 460.167,Z 501.659,A -85,B 0,C 180,E1 -8391.41,E2 -8391.41} C_VEL
LIN {X 0,Y 460.803,Z 485.466,A -85,B 0,C 180,E1 -8391.853,E2 -8391.853} C_VEL
LIN {X 0,Y 462.747,Z 346.784,A -85,B 0,C 180,E1 -8394.106,E2 -8394.106} C_VEL
LIN {X 0,Y 461.542,Z 339.156,A -85,B 0,C 180,E1 -8394.301,E2 -8394.301} C_VEL
LIN {X 0,Y 457.675,Z 319.061,A -85,B 0,C 180,E1 -8394.875,E2 -8394.875} C_VEL
LIN {X 0,Y 458.579,Z 303.374,A -85,B 0,C 180,E1 -8397.266,E2 -8397.266} C_VEL
LIN {X 0,Y 455.594,Z 290.008,A -85,B 0,C 180,E1 -8399.579,E2 -8399.579} C_VEL
LIN {X 0,Y 453.514,Z 281.616,A -85,B 0,C 180,E1 -8401.124,E2 -8401.124} C_VEL
LIN {X 0,Y 453.467,Z 281.626,A -85,B 0,C 180,E1 -8403.913,E2 -8403.913} C_VEL
LIN {X 0,Y 453.44,Z 281.629,A -85,B 0,C 180,E1 -8407.19,E2 -8407.19} C_VEL
LIN {X 0,Y 453.47,Z 281.622,A -85,B 0,C 180,E1 -8410.611,E2 -8410.611} C_VEL
LIN {X 0,Y 453.481,Z 281.623,A -85,B 0,C 180,E1 -8414.527,E2 -8414.527} C_VEL
LIN {X 0,Y 453.439,Z 281.633,A -85,B 0,C 180,E1 -8418.07,E2 -8418.07} C_VEL
LIN {X 0,Y 453.437,Z 281.622,A -85,B 0,C 180,E1 -8420.801,E2 -8420.801} C_VEL
LIN {X 0,Y 453.439,Z 281.63,A -85,B 0,C 180,E1 -8423.915,E2 -8423.915} C_VEL
LIN {X 0,Y 453.472,Z 281.619,A -85,B 0,C 180,E1 -8427.149,E2 -8427.149} C_VEL
LIN {X 0,Y 453.462,Z 281.625,A -85,B 0,C 180,E1 -8430.266,E2 -8430.266} C_VEL
LIN {X 0,Y 453.436,Z 281.624,A -85,B 0,C 180,E1 -8433.288,E2 -8433.288} C_VEL
LIN {X 0,Y 453.489,Z 281.62,A -85,B 0,C 180,E1 -8436.237,E2 -8436.237} C_VEL
LIN {X 0,Y 453.478,Z 281.623,A -85,B 0,C 180,E1 -8439.116,E2 -8439.116} C_VEL
LIN {X 0,Y 453.494,Z 281.625,A -85,B 0,C 180,E1 -8441.943,E2 -8441.943} C_VEL
LIN {X 0,Y 453.529,Z 281.611,A -85,B 0,C 180,E1 -8444.725,E2 -8444.725} C_VEL
LIN {X 0,Y 453.537,Z 281.602,A -85,B 0,C 180,E1 -8448.377,E2 -8448.377} C_VEL
LIN {X 0,Y 453.548,Z 281.61,A -85,B 0,C 180,E1 -8451.084,E2 -8451.084} C_VEL
LIN {X 0,Y 453.628,Z 281.601,A -85,B 0,C 180,E1 -8453.773,E2 -8453.773} C_VEL
LIN {X 0,Y 453.677,Z 281.581,A -85,B 0,C 180,E1 -8457.335,E2 -8457.335} C_VEL
LIN {X 0,Y 453.737,Z 281.588,A -85,B 0,C 180,E1 -8459.999,E2 -8459.999} C_VEL
LIN {X 0,Y 453.702,Z 281.59,A -85,B 0,C 180,E1 -8462.662,E2 -8462.662} C_VEL
LIN {X 0,Y 453.599,Z 281.585,A -85,B 0,C 180,E1 -8466.225,E2 -8466.225} C_VEL
LIN {X 0,Y 453.547,Z 281.604,A -85,B 0,C 180,E1 -8468.913,E2 -8468.913} C_VEL
LIN {X 0,Y 453.555,Z 281.609,A -85,B 0,C 180,E1 -8472.527,E2 -8472.527} C_VEL
LIN {X 0,Y 453.527,Z 281.596,A -85,B 0,C 180,E1 -8476.195,E2 -8476.195} C_VEL
LIN {X 0,Y 453.506,Z 281.608,A -85,B 0,C 180,E1 -8479.038,E2 -8479.038} C_VEL
LIN {X 0,Y 453.464,Z 281.622,A -85,B 0,C 180,E1 -8481.835,E2 -8481.835} C_VEL
LIN {X 0,Y 453.455,Z 281.62,A -85,B 0,C 180,E1 -8484.736,E2 -8484.736} C_VEL
LIN {X 0,Y 453.449,Z 281.611,A -85,B 0,C 180,E1 -8487.941,E2 -8487.941} C_VEL
LIN {X 0,Y 453.452,Z 281.622,A -85,B 0,C 180,E1 -8490.759,E2 -8490.759} C_VEL
LIN {X 0,Y 453.452,Z 281.619,A -85,B 0,C 180,E1 -8493.912,E2 -8493.912} C_VEL
LIN {X 0,Y 453.434,Z 281.615,A -85,B 0,C 180,E1 -8497.189,E2 -8497.189} C_VEL
LIN {X 0,Y 453.455,Z 281.624,A -85,B 0,C 180,E1 -8500.61,E2 -8500.61} C_VEL
LIN {X 0,Y 453.442,Z 281.617,A -85,B 0,C 180,E1 -8504.221,E2 -8504.221} C_VEL
LIN {X 0,Y 453.432,Z 281.624,A -85,B 0,C 180,E1 -8507.002,E2 -8507.002} C_VEL
LIN {X 0,Y 453.477,Z 281.623,A -85,B 0,C 180,E1 -8509.408,E2 -8509.408} C_VEL
LIN {X 0,Y 453.432,Z 281.62,A -85,B 0,C 180,E1 -8512.226,E2 -8512.226} C_VEL
LIN {X 0,Y 453.465,Z 281.626,A -85,B 0,C 180,E1 -8515.223,E2 -8515.223} C_VEL
LIN {X 0,Y 453.447,Z 281.624,A -85,B 0,C 180,E1 -8518.474,E2 -8518.474} C_VEL
LIN {X 0,Y 453.513,Z 281.615,A -85,B 0,C 180,E1 -8522.04,E2 -8522.04} C_VEL
LIN {X 0,Y 453.482,Z 281.619,A -85,B 0,C 180,E1 -8525.264,E2 -8525.264} C_VEL
LIN {X 0,Y 453.462,Z 281.626,A -85,B 0,C 180,E1 -8528.414,E2 -8528.414} C_VEL
LIN {X 0,Y 453.504,Z 281.622,A -85,B 0,C 180,E1 -8531.008,E2 -8531.008} C_VEL
LIN {X 0,Y 453.55,Z 281.607,A -85,B 0,C 180,E1 -8533.879,E2 -8533.879} C_VEL
LIN {X 0,Y 453.584,Z 281.607,A -85,B 0,C 180,E1 -8537.472,E2 -8537.472} C_VEL
LIN {X 0,Y 453.574,Z 281.61,A -85,B 0,C 180,E1 -8541.086,E2 -8541.086} C_VEL
LIN {X 0,Y 453.609,Z 281.607,A -85,B 0,C 180,E1 -8543.032,E2 -8543.032} C_VEL
LIN {X 0,Y 452.921,Z 281.69,A -85,B 0,C 180,E1 -8543.773,E2 -8543.773} C_VEL
LIN {X 0,Y 449.976,Z 282.061,A -85,B 0,C 180,E1 -8544.975,E2 -8544.975} C_VEL
LIN {X 0,Y 447.551,Z 282.362,A -85,B 0,C 180,E1 -8545.945,E2 -8545.945} C_VEL
LIN {X 0,Y 446.604,Z 282.484,A -85,B 0,C 180,E1 -8546.696,E2 -8546.696} C_VEL
LIN {X 0,Y 446.578,Z 282.482,A -85,B 0,C 180,E1 -8546.949,E2 -8546.949} C_VEL
LIN {X 0,Y 446.774,Z 282.464,A -85,B 0,C 180,E1 -8550,E2 -8550} C_VEL
LIN {X 0,Y 446.663,Z 282.55,A -85,B 0,C 180,E1 -8552.085,E2 -8552.085} C_VEL
LIN {X 0,Y 449.638,Z 295.908,A -85,B 0,C 180,E1 -8554.735,E2 -8554.735} C_VEL
LIN {X 0,Y 453.537,Z 306.217,A -85,B 0,C 180,E1 -8555.15,E2 -8555.15} C_VEL
LIN {X 0,Y 456.458,Z 319.584,A -85,B 0,C 180,E1 -8555.549,E2 -8555.549} C_VEL
LIN {X 0,Y 454.359,Z 460.996,A -85,B 0,C 180,E1 -8557.883,E2 -8557.883} C_VEL
LIN {X 0,Y 453.872,Z 476.523,A -85,B 0,C 180,E1 -8558.318,E2 -8558.318} C_VEL
LIN {X 0,Y 453.15,Z 491.496,A -85,B 0,C 180,E1 -8558.922,E2 -8558.922} C_VEL
LIN {X 0,Y 452.341,Z 506.404,A -85,B 0,C 180,E1 -8559.727,E2 -8559.727} C_VEL
LIN {X 0,Y 451.403,Z 520.019,A -85,B 0,C 180,E1 -8560.654,E2 -8560.654} C_VEL
LIN {X 0,Y 450.368,Z 533.811,A -85,B 0,C 180,E1 -8561.818,E2 -8561.818} C_VEL
LIN {X 0,Y 449.401,Z 546.302,A -85,B 0,C 180,E1 -8563.106,E2 -8563.106} C_VEL
LIN {X 0,Y 448.44,Z 557.722,A -85,B 0,C 180,E1 -8564.521,E2 -8564.521} C_VEL
LIN {X 0,Y 447.621,Z 567.384,A -85,B 0,C 180,E1 -8565.947,E2 -8565.947} C_VEL
LIN {X 0,Y 446.87,Z 576.813,A -85,B 0,C 180,E1 -8567.622,E2 -8567.622} C_VEL
LIN {X 0,Y 446.353,Z 584.624,A -85,B 0,C 180,E1 -8569.308,E2 -8569.308} C_VEL
LIN {X 0,Y 445.978,Z 590.189,A -85,B 0,C 180,E1 -8570.766,E2 -8570.766} C_VEL
LIN {X 0,Y 445.752,Z 594.882,A -85,B 0,C 180,E1 -8572.234,E2 -8572.234} C_VEL
LIN {X 0,Y 445.533,Z 599.766,A -85,B 0,C 180,E1 -8574.212,E2 -8574.212} C_VEL
LIN {X 0,Y 445.276,Z 603.215,A -85,B 0,C 180,E1 -8576.226,E2 -8576.226} C_VEL
LIN {X 0,Y 445.185,Z 605.222,A -85,B 0,C 180,E1 -8578.267,E2 -8578.267} C_VEL
LIN {X 0,Y 445.215,Z 605.765,A -85,B 0,C 180,E1 -8579.754,E2 -8579.754} C_VEL
LIN {X 0,Y 445.229,Z 605.408,A -85,B 0,C 180,E1 -8581.531,E2 -8581.531} C_VEL
LIN {X 0,Y 445.251,Z 603.7,A -85,B 0,C 180,E1 -8583.534,E2 -8583.534} C_VEL
LIN {X 0,Y 445.375,Z 601.791,A -85,B 0,C 180,E1 -8584.864,E2 -8584.864} C_VEL
LIN {X 0,Y 445.614,Z 597.768,A -85,B 0,C 180,E1 -8586.82,E2 -8586.82} C_VEL
LIN {X 0,Y 445.859,Z 593.087,A -85,B 0,C 180,E1 -8588.506,E2 -8588.506} C_VEL
LIN {X 0,Y 446.241,Z 587.112,A -85,B 0,C 180,E1 -8590.218,E2 -8590.218} C_VEL
LIN {X 0,Y 446.719,Z 580.101,A -85,B 0,C 180,E1 -8591.855,E2 -8591.855} C_VEL
LIN {X 0,Y 447.305,Z 572.022,A -85,B 0,C 180,E1 -8593.423,E2 -8593.423} C_VEL
LIN {X 0,Y 448.074,Z 562.933,A -85,B 0,C 180,E1 -8594.894,E2 -8594.894} C_VEL
LIN {X 0,Y 449.033,Z 551.195,A -85,B 0,C 180,E1 -8596.479,E2 -8596.479} C_VEL
LIN {X 0,Y 450.071,Z 539.099,A -85,B 0,C 180,E1 -8597.823,E2 -8597.823} C_VEL
LIN {X 0,Y 451.124,Z 525.755,A -85,B 0,C 180,E1 -8599.045,E2 -8599.045} C_VEL
LIN {X 0,Y 452.065,Z 512.77,A -85,B 0,C 180,E1 -8600.021,E2 -8600.021} C_VEL
LIN {X 0,Y 452.95,Z 498.594,A -85,B 0,C 180,E1 -8600.876,E2 -8600.876} C_VEL
LIN {X 0,Y 453.788,Z 483.249,A -85,B 0,C 180,E1 -8601.582,E2 -8601.582} C_VEL
LIN {X 0,Y 454.375,Z 468.596,A -85,B 0,C 180,E1 -8602.075,E2 -8602.075} C_VEL
LIN {X 0,Y 454.729,Z 453.769,A -85,B 0,C 180,E1 -8602.402,E2 -8602.402} C_VEL
LIN {X 0,Y 456.722,Z 319.588,A -85,B 0,C 180,E1 -8604.616,E2 -8604.616} C_VEL
LIN {X 0,Y 453.225,Z 304.752,A -85,B 0,C 180,E1 -8605.092,E2 -8605.092} C_VEL
LIN {X 0,Y 449.777,Z 296.529,A -85,B 0,C 180,E1 -8605.467,E2 -8605.467} C_VEL
LIN {X 0,Y 446.821,Z 284.098,A -85,B 0,C 180,E1 -8608.005,E2 -8608.005} C_VEL
LIN {X 0,Y 446.429,Z 282.502,A -85,B 0,C 180,E1 -8608.374,E2 -8608.374} C_VEL
LIN {X 0,Y 446.468,Z 282.498,A -85,B 0,C 180,E1 -8611.822,E2 -8611.822} C_VEL
LIN {X 0,Y 446.442,Z 282.5,A -85,B 0,C 180,E1 -8614.849,E2 -8614.849} C_VEL
LIN {X 0,Y 446.432,Z 282.499,A -85,B 0,C 180,E1 -8618.246,E2 -8618.246} C_VEL
LIN {X 0,Y 446.443,Z 282.502,A -85,B 0,C 180,E1 -8621.651,E2 -8621.651} C_VEL
LIN {X 0,Y 446.493,Z 282.493,A -85,B 0,C 180,E1 -8624.481,E2 -8624.481} C_VEL
LIN {X 0,Y 446.503,Z 282.49,A -85,B 0,C 180,E1 -8628.194,E2 -8628.194} C_VEL
LIN {X 0,Y 446.587,Z 282.478,A -85,B 0,C 180,E1 -8631.859,E2 -8631.859} C_VEL
LIN {X 0,Y 446.627,Z 282.473,A -85,B 0,C 180,E1 -8634.584,E2 -8634.584} C_VEL
LIN {X 0,Y 446.653,Z 282.471,A -85,B 0,C 180,E1 -8638.198,E2 -8638.198} C_VEL
LIN {X 0,Y 446.78,Z 282.454,A -85,B 0,C 180,E1 -8640.001,E2 -8640.001} C_VEL
LIN {X 0,Y 446.676,Z 282.469,A -85,B 0,C 180,E1 -8642.707,E2 -8642.707} C_VEL
LIN {X 0,Y 446.618,Z 282.476,A -85,B 0,C 180,E1 -8646.325,E2 -8646.325} C_VEL
LIN {X 0,Y 446.521,Z 282.491,A -85,B 0,C 180,E1 -8649.057,E2 -8649.057} C_VEL
LIN {X 0,Y 446.512,Z 282.493,A -85,B 0,C 180,E1 -8652.731,E2 -8652.731} C_VEL
LIN {X 0,Y 446.48,Z 282.496,A -85,B 0,C 180,E1 -8656.461,E2 -8656.461} C_VEL
LIN {X 0,Y 446.46,Z 282.493,A -85,B 0,C 180,E1 -8659.305,E2 -8659.305} C_VEL
LIN {X 0,Y 446.408,Z 282.505,A -85,B 0,C 180,E1 -8662.201,E2 -8662.201} C_VEL
LIN {X 0,Y 446.406,Z 282.5,A -85,B 0,C 180,E1 -8665.157,E2 -8665.157} C_VEL
LIN {X 0,Y 446.431,Z 282.502,A -85,B 0,C 180,E1 -8668.183,E2 -8668.183} C_VEL
LIN {X 0,Y 446.401,Z 282.498,A -85,B 0,C 180,E1 -8671.303,E2 -8671.303} C_VEL
LIN {X 0,Y 446.413,Z 282.502,A -85,B 0,C 180,E1 -8674.525,E2 -8674.525} C_VEL
LIN {X 0,Y 446.391,Z 282.507,A -85,B 0,C 180,E1 -8678.077,E2 -8678.077} C_VEL
LIN {X 0,Y 446.394,Z 282.501,A -85,B 0,C 180,E1 -8681.396,E2 -8681.396} C_VEL
LIN {X 0,Y 446.416,Z 282.5,A -85,B 0,C 180,E1 -8685.109,E2 -8685.109} C_VEL
LIN {X 0,Y 446.396,Z 282.505,A -85,B 0,C 180,E1 -8688.607,E2 -8688.607} C_VEL
LIN {X 0,Y 446.395,Z 282.508,A -85,B 0,C 180,E1 -8691.925,E2 -8691.925} C_VEL
LIN {X 0,Y 446.419,Z 282.499,A -85,B 0,C 180,E1 -8695.477,E2 -8695.477} C_VEL
LIN {X 0,Y 446.446,Z 282.597,A -85,B 0,C 180,E1 -8698.463,E2 -8698.463} C_VEL
LIN {X 0,Y 449.959,Z 296.433,A -85,B 0,C 180,E1 -8701.041,E2 -8701.041} C_VEL
LIN {X 0,Y 451.796,Z 305.708,A -85,B 0,C 180,E1 -8702.673,E2 -8702.673} C_VEL
LIN {X 0,Y 450.914,Z 318.315,A -85,B 0,C 180,E1 -8704.635,E2 -8704.635} C_VEL
LIN {X 0,Y 456.425,Z 346.561,A -85,B 0,C 180,E1 -8705.478,E2 -8705.478} C_VEL
LIN {X 0,Y 454.362,Z 484.233,A -85,B 0,C 180,E1 -8707.761,E2 -8707.761} C_VEL
LIN {X 0,Y 453.764,Z 500.226,A -85,B 0,C 180,E1 -8708.197,E2 -8708.197} C_VEL
LIN {X 0,Y 452.944,Z 515.479,A -85,B 0,C 180,E1 -8708.804,E2 -8708.804} C_VEL
LIN {X 0,Y 452.067,Z 529.173,A -85,B 0,C 180,E1 -8709.526,E2 -8709.526} C_VEL
LIN {X 0,Y 451.16,Z 542.804,A -85,B 0,C 180,E1 -8710.433,E2 -8710.433} C_VEL
LIN {X 0,Y 450.01,Z 556.659,A -85,B 0,C 180,E1 -8711.564,E2 -8711.564} C_VEL
LIN {X 0,Y 449.038,Z 569.231,A -85,B 0,C 180,E1 -8712.821,E2 -8712.821} C_VEL
LIN {X 0,Y 448.151,Z 579.73,A -85,B 0,C 180,E1 -8714.072,E2 -8714.072} C_VEL
LIN {X 0,Y 447.422,Z 589.502,A -85,B 0,C 180,E1 -8715.445,E2 -8715.445} C_VEL
LIN {X 0,Y 446.675,Z 599.095,A -85,B 0,C 180,E1 -8717.044,E2 -8717.044} C_VEL
LIN {X 0,Y 446.269,Z 607.095,A -85,B 0,C 180,E1 -8718.648,E2 -8718.648} C_VEL
LIN {X 0,Y 445.771,Z 614.561,A -85,B 0,C 180,E1 -8720.472,E2 -8720.472} C_VEL
LIN {X 0,Y 445.564,Z 620.491,A -85,B 0,C 180,E1 -8722.296,E2 -8722.296} C_VEL
LIN {X 0,Y 445.376,Z 624.337,A -85,B 0,C 180,E1 -8723.795,E2 -8723.795} C_VEL
LIN {X 0,Y 445.364,Z 627.58,A -85,B 0,C 180,E1 -8725.475,E2 -8725.475} C_VEL
LIN {X 0,Y 445.42,Z 629.931,A -85,B 0,C 180,E1 -8727.287,E2 -8727.287} C_VEL
LIN {X 0,Y 445.337,Z 631.114,A -85,B 0,C 180,E1 -8729.096,E2 -8729.096} C_VEL
LIN {X 0,Y 445.337,Z 631.123,A -85,B 0,C 180,E1 -8730.905,E2 -8730.905} C_VEL
LIN {X 0,Y 445.42,Z 629.947,A -85,B 0,C 180,E1 -8732.713,E2 -8732.713} C_VEL
LIN {X 0,Y 445.365,Z 627.604,A -85,B 0,C 180,E1 -8734.526,E2 -8734.526} C_VEL
LIN {X 0,Y 445.434,Z 624.05,A -85,B 0,C 180,E1 -8736.341,E2 -8736.341} C_VEL
LIN {X 0,Y 445.611,Z 619.193,A -85,B 0,C 180,E1 -8738.161,E2 -8738.161} C_VEL
LIN {X 0,Y 445.838,Z 612.898,A -85,B 0,C 180,E1 -8739.986,E2 -8739.986} C_VEL
LIN {X 0,Y 446.284,Z 606.108,A -85,B 0,C 180,E1 -8741.583,E2 -8741.583} C_VEL
LIN {X 0,Y 446.789,Z 597.877,A -85,B 0,C 180,E1 -8743.184,E2 -8743.184} C_VEL
LIN {X 0,Y 447.507,Z 588.005,A -85,B 0,C 180,E1 -8744.786,E2 -8744.786} C_VEL
LIN {X 0,Y 448.345,Z 577.898,A -85,B 0,C 180,E1 -8746.155,E2 -8746.155} C_VEL
LIN {X 0,Y 449.305,Z 566.104,A -85,B 0,C 180,E1 -8747.5,E2 -8747.5} C_VEL
LIN {X 0,Y 450.223,Z 553.884,A -85,B 0,C 180,E1 -8748.663,E2 -8748.663} C_VEL
LIN {X 0,Y 451.239,Z 540.893,A -85,B 0,C 180,E1 -8749.682,E2 -8749.682} C_VEL
LIN {X 0,Y 452.173,Z 526.664,A -85,B 0,C 180,E1 -8750.588,E2 -8750.588} C_VEL
LIN {X 0,Y 453.062,Z 512.206,A -85,B 0,C 180,E1 -8751.305,E2 -8751.305} C_VEL
LIN {X 0,Y 453.732,Z 497.463,A -85,B 0,C 180,E1 -8751.853,E2 -8751.853} C_VEL
LIN {X 0,Y 454.244,Z 481.744,A -85,B 0,C 180,E1 -8752.245,E2 -8752.245} C_VEL
LIN {X 0,Y 456.234,Z 347.722,A -85,B 0,C 180,E1 -8754.444,E2 -8754.444} C_VEL
LIN {X 0,Y 455.234,Z 341.264,A -85,B 0,C 180,E1 -8754.611,E2 -8754.611} C_VEL
LIN {X 0,Y 450.916,Z 318.894,A -85,B 0,C 180,E1 -8755.26,E2 -8755.26} C_VEL
LIN {X 0,Y 451.766,Z 305.577,A -85,B 0,C 180,E1 -8757.319,E2 -8757.319} C_VEL
LIN {X 0,Y 449.443,Z 294.486,A -85,B 0,C 180,E1 -8759.252,E2 -8759.252} C_VEL
LIN {X 0,Y 446.427,Z 282.502,A -85,B 0,C 180,E1 -8761.474,E2 -8761.474} C_VEL
LIN {X 0,Y 446.423,Z 282.506,A -85,B 0,C 180,E1 -8764.523,E2 -8764.523} C_VEL
LIN {X 0,Y 446.4,Z 282.506,A -85,B 0,C 180,E1 -8768.076,E2 -8768.076} C_VEL
LIN {X 0,Y 446.4,Z 282.502,A -85,B 0,C 180,E1 -8771.394,E2 -8771.394} C_VEL
LIN {X 0,Y 446.421,Z 282.5,A -85,B 0,C 180,E1 -8775.107,E2 -8775.107} C_VEL
LIN {X 0,Y 446.402,Z 282.506,A -85,B 0,C 180,E1 -8778.605,E2 -8778.605} C_VEL
LIN {X 0,Y 446.396,Z 282.506,A -85,B 0,C 180,E1 -8781.923,E2 -8781.923} C_VEL
LIN {X 0,Y 446.418,Z 282.496,A -85,B 0,C 180,E1 -8785.475,E2 -8785.475} C_VEL
LIN {X 0,Y 446.41,Z 282.5,A -85,B 0,C 180,E1 -8788.698,E2 -8788.698} C_VEL
LIN {X 0,Y 446.422,Z 282.504,A -85,B 0,C 180,E1 -8791.835,E2 -8791.835} C_VEL
LIN {X 0,Y 446.416,Z 282.501,A -85,B 0,C 180,E1 -8794.844,E2 -8794.844} C_VEL
LIN {X 0,Y 446.445,Z 282.5,A -85,B 0,C 180,E1 -8798.244,E2 -8798.244} C_VEL
LIN {X 0,Y 446.444,Z 282.501,A -85,B 0,C 180,E1 -8801.647,E2 -8801.647} C_VEL
LIN {X 0,Y 446.49,Z 282.488,A -85,B 0,C 180,E1 -8804.478,E2 -8804.478} C_VEL
LIN {X 0,Y 446.5,Z 282.479,A -85,B 0,C 180,E1 -8808.191,E2 -8808.191} C_VEL
LIN {X 0,Y 446.499,Z 282.487,A -85,B 0,C 180,E1 -8810.943,E2 -8810.943} C_VEL
LIN {X 0,Y 446.598,Z 282.478,A -85,B 0,C 180,E1 -8813.674,E2 -8813.674} C_VEL
LIN {X 0,Y 446.629,Z 282.458,A -85,B 0,C 180,E1 -8817.293,E2 -8817.293} C_VEL
LIN {X 0,Y 446.688,Z 282.466,A -85,B 0,C 180,E1 -8819.999,E2 -8819.999} C_VEL
LIN {X 0,Y 446.652,Z 282.469,A -85,B 0,C 180,E1 -8822.704,E2 -8822.704} C_VEL
LIN {X 0,Y 446.57,Z 282.459,A -85,B 0,C 180,E1 -8826.323,E2 -8826.323} C_VEL
LIN {X 0,Y 446.498,Z 282.483,A -85,B 0,C 180,E1 -8829.054,E2 -8829.054} C_VEL
LIN {X 0,Y 446.512,Z 282.487,A -85,B 0,C 180,E1 -8832.728,E2 -8832.728} C_VEL
LIN {X 0,Y 446.473,Z 282.474,A -85,B 0,C 180,E1 -8836.458,E2 -8836.458} C_VEL
LIN {X 0,Y 446.457,Z 282.49,A -85,B 0,C 180,E1 -8839.302,E2 -8839.302} C_VEL
LIN {X 0,Y 446.404,Z 282.5,A -85,B 0,C 180,E1 -8842.198,E2 -8842.198} C_VEL
LIN {X 0,Y 446.407,Z 282.496,A -85,B 0,C 180,E1 -8845.153,E2 -8845.153} C_VEL
LIN {X 0,Y 446.403,Z 282.488,A -85,B 0,C 180,E1 -8848.182,E2 -8848.182} C_VEL
LIN {X 0,Y 446.398,Z 282.508,A -85,B 0,C 180,E1 -8851.299,E2 -8851.299} C_VEL
LIN {X 0,Y 446.407,Z 282.497,A -85,B 0,C 180,E1 -8854.522,E2 -8854.522} C_VEL
LIN {X 0,Y 446.395,Z 282.493,A -85,B 0,C 180,E1 -8858.077,E2 -8858.077} C_VEL
LIN {X 0,Y 446.391,Z 282.506,A -85,B 0,C 180,E1 -8861.392,E2 -8861.392} C_VEL
LIN {X 0,Y 446.405,Z 282.494,A -85,B 0,C 180,E1 -8864.891,E2 -8864.891} C_VEL
LIN {X 0,Y 446.405,Z 282.501,A -85,B 0,C 180,E1 -8867.724,E2 -8867.724} C_VEL
LIN {X 0,Y 446.422,Z 282.501,A -85,B 0,C 180,E1 -8870.971,E2 -8870.971} C_VEL
LIN {X 0,Y 446.401,Z 282.497,A -85,B 0,C 180,E1 -8874.373,E2 -8874.373} C_VEL
LIN {X 0,Y 446.402,Z 282.5,A -85,B 0,C 180,E1 -8877.637,E2 -8877.637} C_VEL
LIN {X 0,Y 446.429,Z 282.496,A -85,B 0,C 180,E1 -8880.79,E2 -8880.79} C_VEL
LIN {X 0,Y 446.461,Z 282.491,A -85,B 0,C 180,E1 -8883.848,E2 -8883.848} C_VEL
LIN {X 0,Y 446.408,Z 282.506,A -85,B 0,C 180,E1 -8886.822,E2 -8886.822} C_VEL
LIN {X 0,Y 446.425,Z 282.494,A -85,B 0,C 180,E1 -8889.736,E2 -8889.736} C_VEL
LIN {X 0,Y 446.444,Z 282.501,A -85,B 0,C 180,E1 -8892.596,E2 -8892.596} C_VEL
LIN {X 0,Y 446.451,Z 282.496,A -85,B 0,C 180,E1 -8895.412,E2 -8895.412} C_VEL
LIN {X 0,Y 446.523,Z 282.489,A -85,B 0,C 180,E1 -8898.193,E2 -8898.193} C_VEL
LIN {X 0,Y 446.582,Z 282.479,A -85,B 0,C 180,E1 -8901.857,E2 -8901.857} C_VEL
LIN {X 0,Y 446.621,Z 282.478,A -85,B 0,C 180,E1 -8904.582,E2 -8904.582} C_VEL
LIN {X 0,Y 446.578,Z 282.482,A -85,B 0,C 180,E1 -8906.949,E2 -8906.949} C_VEL
LIN {X 0,Y 446.054,Z 282.549,A -85,B 0,C 180,E1 -8907.702,E2 -8907.702} C_VEL
LIN {X 0,Y 443.26,Z 282.901,A -85,B 0,C 180,E1 -8908.926,E2 -8908.926} C_VEL
LIN {X 0,Y 440.798,Z 283.21,A -85,B 0,C 180,E1 -8909.914,E2 -8909.914} C_VEL
LIN {X 0,Y 439.717,Z 283.344,A -85,B 0,C 180,E1 -8910.677,E2 -8910.677} C_VEL
LIN {X 0,Y 439.62,Z 283.356,A -85,B 0,C 180,E1 -8910.936,E2 -8910.936} C_VEL
LIN {X 0,Y 439.617,Z 283.433,A -85,B 0,C 180,E1 -8911.746,E2 -8911.746} C_VEL
LIN {X 0,Y 442.464,Z 296.306,A -85,B 0,C 180,E1 -8914.318,E2 -8914.318} C_VEL
LIN {X 0,Y 447.332,Z 308.557,A -85,B 0,C 180,E1 -8914.83,E2 -8914.83} C_VEL
LIN {X 0,Y 449.971,Z 320.293,A -85,B 0,C 180,E1 -8915.191,E2 -8915.191} C_VEL
LIN {X 0,Y 447.77,Z 461.138,A -85,B 0,C 180,E1 -8917.553,E2 -8917.553} C_VEL
LIN {X 0,Y 447.207,Z 477.216,A -85,B 0,C 180,E1 -8918.012,E2 -8918.012} C_VEL
LIN {X 0,Y 446.423,Z 492.736,A -85,B 0,C 180,E1 -8918.658,E2 -8918.658} C_VEL
LIN {X 0,Y 445.656,Z 506.506,A -85,B 0,C 180,E1 -8919.416,E2 -8919.416} C_VEL
LIN {X 0,Y 444.668,Z 520.154,A -85,B 0,C 180,E1 -8920.356,E2 -8920.356} C_VEL
LIN {X 0,Y 443.632,Z 533.595,A -85,B 0,C 180,E1 -8921.502,E2 -8921.502} C_VEL
LIN {X 0,Y 442.635,Z 545.462,A -85,B 0,C 180,E1 -8922.726,E2 -8922.726} C_VEL
LIN {X 0,Y 441.632,Z 556.847,A -85,B 0,C 180,E1 -8924.134,E2 -8924.134} C_VEL
LIN {X 0,Y 440.679,Z 567.573,A -85,B 0,C 180,E1 -8925.73,E2 -8925.73} C_VEL
LIN {X 0,Y 439.91,Z 576.997,A -85,B 0,C 180,E1 -8927.43,E2 -8927.43} C_VEL
LIN {X 0,Y 439.295,Z 585.407,A -85,B 0,C 180,E1 -8929.29,E2 -8929.29} C_VEL
LIN {X 0,Y 438.816,Z 592.08,A -85,B 0,C 180,E1 -8931.121,E2 -8931.121} C_VEL
LIN {X 0,Y 438.567,Z 597.707,A -85,B 0,C 180,E1 -8933.116,E2 -8933.116} C_VEL
LIN {X 0,Y 438.364,Z 600.954,A -85,B 0,C 180,E1 -8934.634,E2 -8934.634} C_VEL
LIN {X 0,Y 438.174,Z 604.044,A -85,B 0,C 180,E1 -8936.685,E2 -8936.685} C_VEL
LIN {X 0,Y 438.087,Z 605.7,A -85,B 0,C 180,E1 -8938.768,E2 -8938.768} C_VEL
LIN {X 0,Y 438.12,Z 606.009,A -85,B 0,C 180,E1 -8939.982,E2 -8939.982} C_VEL
LIN {X 0,Y 438.13,Z 605.409,A -85,B 0,C 180,E1 -8941.96,E2 -8941.96} C_VEL
LIN {X 0,Y 438.178,Z 604.032,A -85,B 0,C 180,E1 -8943.489,E2 -8943.489} C_VEL
LIN {X 0,Y 438.328,Z 601.486,A -85,B 0,C 180,E1 -8945.253,E2 -8945.253} C_VEL
LIN {X 0,Y 438.525,Z 598.4,A -85,B 0,C 180,E1 -8946.747,E2 -8946.747} C_VEL
LIN {X 0,Y 438.813,Z 593.278,A -85,B 0,C 180,E1 -8948.653,E2 -8948.653} C_VEL
LIN {X 0,Y 439.219,Z 587.296,A -85,B 0,C 180,E1 -8950.393,E2 -8950.393} C_VEL
LIN {X 0,Y 439.775,Z 579.79,A -85,B 0,C 180,E1 -8952.158,E2 -8952.158} C_VEL
LIN {X 0,Y 440.492,Z 570.628,A -85,B 0,C 180,E1 -8953.918,E2 -8953.918} C_VEL
LIN {X 0,Y 441.403,Z 560.44,A -85,B 0,C 180,E1 -8955.531,E2 -8955.531} C_VEL
LIN {X 0,Y 442.38,Z 549.672,A -85,B 0,C 180,E1 -8956.951,E2 -8956.951} C_VEL
LIN {X 0,Y 443.409,Z 537.723,A -85,B 0,C 180,E1 -8958.267,E2 -8958.267} C_VEL
LIN {X 0,Y 444.431,Z 525.606,A -85,B 0,C 180,E1 -8959.378,E2 -8959.378} C_VEL
LIN {X 0,Y 445.455,Z 512.143,A -85,B 0,C 180,E1 -8960.393,E2 -8960.393} C_VEL
LIN {X 0,Y 446.431,Z 497.689,A -85,B 0,C 180,E1 -8961.259,E2 -8961.259} C_VEL
LIN {X 0,Y 447.226,Z 483.22,A -85,B 0,C 180,E1 -8961.929,E2 -8961.929} C_VEL
LIN {X 0,Y 447.837,Z 468.391,A -85,B 0,C 180,E1 -8962.43,E2 -8962.43} C_VEL
LIN {X 0,Y 448.222,Z 453.227,A -85,B 0,C 180,E1 -8962.763,E2 -8962.763} C_VEL
LIN {X 0,Y 450.276,Z 320.108,A -85,B 0,C 180,E1 -8965.001,E2 -8965.001} C_VEL
LIN {X 0,Y 447.247,Z 307.718,A -85,B 0,C 180,E1 -8965.415,E2 -8965.415} C_VEL
LIN {X 0,Y 442.633,Z 296.787,A -85,B 0,C 180,E1 -8965.92,E2 -8965.92} C_VEL
LIN {X 0,Y 439.717,Z 284.755,A -85,B 0,C 180,E1 -8968.439,E2 -8968.439} C_VEL
LIN {X 0,Y 439.377,Z 283.382,A -85,B 0,C 180,E1 -8968.747,E2 -8968.747} C_VEL
LIN {X 0,Y 439.428,Z 283.374,A -85,B 0,C 180,E1 -8972.369,E2 -8972.369} C_VEL
LIN {X 0,Y 439.399,Z 283.378,A -85,B 0,C 180,E1 -8975.736,E2 -8975.736} C_VEL
LIN {X 0,Y 439.374,Z 283.385,A -85,B 0,C 180,E1 -8979.398,E2 -8979.398} C_VEL
LIN {X 0,Y 439.417,Z 283.375,A -85,B 0,C 180,E1 -8982.311,E2 -8982.311} C_VEL
LIN {X 0,Y 439.433,Z 283.374,A -85,B 0,C 180,E1 -8985.175,E2 -8985.175} C_VEL
LIN {X 0,Y 439.469,Z 283.366,A -85,B 0,C 180,E1 -8988.003,E2 -8988.003} C_VEL
LIN {X 0,Y 439.534,Z 283.358,A -85,B 0,C 180,E1 -8991.728,E2 -8991.728} C_VEL
LIN {X 0,Y 439.602,Z 283.348,A -85,B 0,C 180,E1 -8994.497,E2 -8994.497} C_VEL
LIN {X 0,Y 439.623,Z 283.347,A -85,B 0,C 180,E1 -8998.169,E2 -8998.169} C_VEL
LIN {X 0,Y 439.75,Z 283.33,A -85,B 0,C 180,E1 -9000.002,E2 -9000.002} C_VEL
LIN {X 0,Y 439.625,Z 283.348,A -85,B 0,C 180,E1 -9002.75,E2 -9002.75} C_VEL
LIN {X 0,Y 439.589,Z 283.353,A -85,B 0,C 180,E1 -9006.427,E2 -9006.427} C_VEL
LIN {X 0,Y 439.484,Z 283.366,A -85,B 0,C 180,E1 -9009.203,E2 -9009.203} C_VEL
LIN {X 0,Y 439.456,Z 283.369,A -85,B 0,C 180,E1 -9012.939,E2 -9012.939} C_VEL
LIN {X 0,Y 439.438,Z 283.373,A -85,B 0,C 180,E1 -9016.35,E2 -9016.35} C_VEL
LIN {X 0,Y 439.394,Z 283.373,A -85,B 0,C 180,E1 -9019.628,E2 -9019.628} C_VEL
LIN {X 0,Y 439.354,Z 283.382,A -85,B 0,C 180,E1 -9022.577,E2 -9022.577} C_VEL
LIN {X 0,Y 439.354,Z 283.378,A -85,B 0,C 180,E1 -9025.589,E2 -9025.589} C_VEL
LIN {X 0,Y 439.384,Z 283.376,A -85,B 0,C 180,E1 -9028.677,E2 -9028.677} C_VEL
LIN {X 0,Y 439.356,Z 283.378,A -85,B 0,C 180,E1 -9032.03,E2 -9032.03} C_VEL
LIN {X 0,Y 439.38,Z 283.375,A -85,B 0,C 180,E1 -9035.34,E2 -9035.34} C_VEL
LIN {X 0,Y 439.348,Z 283.38,A -85,B 0,C 180,E1 -9038.6,E2 -9038.6} C_VEL
LIN {X 0,Y 439.343,Z 283.385,A -85,B 0,C 180,E1 -9042.212,E2 -9042.212} C_VEL
LIN {X 0,Y 439.37,Z 283.378,A -85,B 0,C 180,E1 -9045.268,E2 -9045.268} C_VEL
LIN {X 0,Y 439.359,Z 283.38,A -85,B 0,C 180,E1 -9048.749,E2 -9048.749} C_VEL
LIN {X 0,Y 439.353,Z 283.385,A -85,B 0,C 180,E1 -9051.612,E2 -9051.612} C_VEL
LIN {X 0,Y 439.39,Z 283.377,A -85,B 0,C 180,E1 -9054.845,E2 -9054.845} C_VEL
LIN {X 0,Y 439.394,Z 283.456,A -85,B 0,C 180,E1 -9058.055,E2 -9058.055} C_VEL
LIN {X 0,Y 442.7,Z 296.341,A -85,B 0,C 180,E1 -9060.52,E2 -9060.52} C_VEL
LIN {X 0,Y 444.998,Z 306.925,A -85,B 0,C 180,E1 -9062.437,E2 -9062.437} C_VEL
LIN {X 0,Y 444.241,Z 318.147,A -85,B 0,C 180,E1 -9064.22,E2 -9064.22} C_VEL
LIN {X 0,Y 449.902,Z 346.9,A -85,B 0,C 180,E1 -9065.095,E2 -9065.095} C_VEL
LIN {X 0,Y 448.757,Z 427.884,A -85,B 0,C 180,E1 -9066.463,E2 -9066.463} C_VEL
LIN {X 0,Y 447.77,Z 485.526,A -85,B 0,C 180,E1 -9067.447,E2 -9067.447} C_VEL
LIN {X 0,Y 447.12,Z 501.079,A -85,B 0,C 180,E1 -9067.892,E2 -9067.892} C_VEL
LIN {X 0,Y 446.345,Z 515.066,A -85,B 0,C 180,E1 -9068.46,E2 -9068.46} C_VEL
LIN {X 0,Y 445.403,Z 529.038,A -85,B 0,C 180,E1 -9069.206,E2 -9069.206} C_VEL
LIN {X 0,Y 444.455,Z 542.653,A -85,B 0,C 180,E1 -9070.126,E2 -9070.126} C_VEL
LIN {X 0,Y 443.234,Z 556.498,A -85,B 0,C 180,E1 -9071.272,E2 -9071.272} C_VEL
LIN {X 0,Y 442.319,Z 567.956,A -85,B 0,C 180,E1 -9072.43,E2 -9072.43} C_VEL
LIN {X 0,Y 441.285,Z 579.547,A -85,B 0,C 180,E1 -9073.818,E2 -9073.818} C_VEL
LIN {X 0,Y 440.484,Z 589.309,A -85,B 0,C 180,E1 -9075.21,E2 -9075.21} C_VEL
LIN {X 0,Y 439.686,Z 598.897,A -85,B 0,C 180,E1 -9076.835,E2 -9076.835} C_VEL
LIN {X 0,Y 439.232,Z 606.896,A -85,B 0,C 180,E1 -9078.463,E2 -9078.463} C_VEL
LIN {X 0,Y 438.7,Z 614.361,A -85,B 0,C 180,E1 -9080.317,E2 -9080.317} C_VEL
LIN {X 0,Y 438.488,Z 620.29,A -85,B 0,C 180,E1 -9082.17,E2 -9082.17} C_VEL
LIN {X 0,Y 438.296,Z 624.404,A -85,B 0,C 180,E1 -9083.808,E2 -9083.808} C_VEL
LIN {X 0,Y 438.286,Z 627.38,A -85,B 0,C 180,E1 -9085.402,E2 -9085.402} C_VEL
LIN {X 0,Y 438.327,Z 629.73,A -85,B 0,C 180,E1 -9087.243,E2 -9087.243} C_VEL
LIN {X 0,Y 438.251,Z 630.911,A -85,B 0,C 180,E1 -9089.082,E2 -9089.082} C_VEL
LIN {X 0,Y 438.251,Z 630.92,A -85,B 0,C 180,E1 -9090.919,E2 -9090.919} C_VEL
LIN {X 0,Y 438.327,Z 629.74,A -85,B 0,C 180,E1 -9092.757,E2 -9092.757} C_VEL
LIN {X 0,Y 438.288,Z 627.394,A -85,B 0,C 180,E1 -9094.599,E2 -9094.599} C_VEL
LIN {X 0,Y 438.36,Z 623.835,A -85,B 0,C 180,E1 -9096.444,E2 -9096.444} C_VEL
LIN {X 0,Y 438.544,Z 618.971,A -85,B 0,C 180,E1 -9098.293,E2 -9098.293} C_VEL
LIN {X 0,Y 438.785,Z 612.667,A -85,B 0,C 180,E1 -9100.148,E2 -9100.148} C_VEL
LIN {X 0,Y 439.233,Z 605.867,A -85,B 0,C 180,E1 -9101.772,E2 -9101.772} C_VEL
LIN {X 0,Y 439.781,Z 597.625,A -85,B 0,C 180,E1 -9103.398,E2 -9103.398} C_VEL
LIN {X 0,Y 440.569,Z 587.738,A -85,B 0,C 180,E1 -9105.024,E2 -9105.024} C_VEL
LIN {X 0,Y 441.468,Z 577.615,A -85,B 0,C 180,E1 -9106.414,E2 -9106.414} C_VEL
LIN {X 0,Y 442.443,Z 565.583,A -85,B 0,C 180,E1 -9107.805,E2 -9107.805} C_VEL
LIN {X 0,Y 443.45,Z 553.561,A -85,B 0,C 180,E1 -9108.959,E2 -9108.959} C_VEL
LIN {X 0,Y 444.521,Z 540.537,A -85,B 0,C 180,E1 -9109.992,E2 -9109.992} C_VEL
LIN {X 0,Y 445.494,Z 526.256,A -85,B 0,C 180,E1 -9110.911,E2 -9110.911} C_VEL
LIN {X 0,Y 446.401,Z 511.723,A -85,B 0,C 180,E1 -9111.639,E2 -9111.639} C_VEL
LIN {X 0,Y 447.11,Z 496.858,A -85,B 0,C 180,E1 -9112.194,E2 -9112.194} C_VEL
LIN {X 0,Y 447.662,Z 480.878,A -85,B 0,C 180,E1 -9112.59,E2 -9112.59} C_VEL
LIN {X 0,Y 449.732,Z 348.185,A -85,B 0,C 180,E1 -9114.8,E2 -9114.8} C_VEL
LIN {X 0,Y 444.164,Z 318.661,A -85,B 0,C 180,E1 -9115.668,E2 -9115.668} C_VEL
LIN {X 0,Y 444.906,Z 306.69,A -85,B 0,C 180,E1 -9117.553,E2 -9117.553} C_VEL
LIN {X 0,Y 441.746,Z 292.605,A -85,B 0,C 180,E1 -9120.076,E2 -9120.076} C_VEL
LIN {X 0,Y 439.371,Z 283.383,A -85,B 0,C 180,E1 -9121.827,E2 -9121.827} C_VEL
LIN {X 0,Y 439.39,Z 283.381,A -85,B 0,C 180,E1 -9125.338,E2 -9125.338} C_VEL
LIN {X 0,Y 439.356,Z 283.385,A -85,B 0,C 180,E1 -9128.597,E2 -9128.597} C_VEL
LIN {X 0,Y 439.348,Z 283.384,A -85,B 0,C 180,E1 -9132.209,E2 -9132.209} C_VEL
LIN {X 0,Y 439.375,Z 283.378,A -85,B 0,C 180,E1 -9135.266,E2 -9135.266} C_VEL
LIN {X 0,Y 439.364,Z 283.382,A -85,B 0,C 180,E1 -9138.746,E2 -9138.746} C_VEL
LIN {X 0,Y 439.354,Z 283.379,A -85,B 0,C 180,E1 -9141.61,E2 -9141.61} C_VEL
LIN {X 0,Y 439.389,Z 283.371,A -85,B 0,C 180,E1 -9144.842,E2 -9144.842} C_VEL
LIN {X 0,Y 439.368,Z 283.382,A -85,B 0,C 180,E1 -9148.138,E2 -9148.138} C_VEL
LIN {X 0,Y 439.398,Z 283.378,A -85,B 0,C 180,E1 -9151.605,E2 -9151.605} C_VEL
LIN {X 0,Y 439.362,Z 283.381,A -85,B 0,C 180,E1 -9154.411,E2 -9154.411} C_VEL
LIN {X 0,Y 439.359,Z 283.381,A -85,B 0,C 180,E1 -9157.423,E2 -9157.423} C_VEL
LIN {X 0,Y 439.438,Z 283.367,A -85,B 0,C 180,E1 -9160.662,E2 -9160.662} C_VEL
LIN {X 0,Y 439.451,Z 283.366,A -85,B 0,C 180,E1 -9164.223,E2 -9164.223} C_VEL
LIN {X 0,Y 439.47,Z 283.352,A -85,B 0,C 180,E1 -9168,E2 -9168} C_VEL
LIN {X 0,Y 439.473,Z 283.37,A -85,B 0,C 180,E1 -9171.723,E2 -9171.723} C_VEL
LIN {X 0,Y 439.589,Z 283.344,A -85,B 0,C 180,E1 -9174.494,E2 -9174.494} C_VEL
LIN {X 0,Y 439.614,Z 283.339,A -85,B 0,C 180,E1 -9178.166,E2 -9178.166} C_VEL
LIN {X 0,Y 439.639,Z 283.344,A -85,B 0,C 180,E1 -9179.998,E2 -9179.998} C_VEL
LIN {X 0,Y 439.603,Z 283.347,A -85,B 0,C 180,E1 -9182.747,E2 -9182.747} C_VEL
LIN {X 0,Y 439.573,Z 283.338,A -85,B 0,C 180,E1 -9185.503,E2 -9185.503} C_VEL
LIN {X 0,Y 439.452,Z 283.357,A -85,B 0,C 180,E1 -9188.274,E2 -9188.274} C_VEL
LIN {X 0,Y 439.416,Z 283.373,A -85,B 0,C 180,E1 -9191.064,E2 -9191.064} C_VEL
LIN {X 0,Y 439.403,Z 283.369,A -85,B 0,C 180,E1 -9193.88,E2 -9193.88} C_VEL
LIN {X 0,Y 439.415,Z 283.354,A -85,B 0,C 180,E1 -9196.73,E2 -9196.73} C_VEL
LIN {X 0,Y 439.39,Z 283.375,A -85,B 0,C 180,E1 -9199.625,E2 -9199.625} C_VEL
LIN {X 0,Y 439.35,Z 283.379,A -85,B 0,C 180,E1 -9202.574,E2 -9202.574} C_VEL
LIN {X 0,Y 439.352,Z 283.367,A -85,B 0,C 180,E1 -9205.586,E2 -9205.586} C_VEL
LIN {X 0,Y 439.369,Z 283.365,A -85,B 0,C 180,E1 -9208.675,E2 -9208.675} C_VEL
LIN {X 0,Y 439.351,Z 283.379,A -85,B 0,C 180,E1 -9212.028,E2 -9212.028} C_VEL
LIN {X 0,Y 439.376,Z 283.366,A -85,B 0,C 180,E1 -9215.338,E2 -9215.338} C_VEL
LIN {X 0,Y 439.347,Z 283.373,A -85,B 0,C 180,E1 -9218.596,E2 -9218.596} C_VEL
LIN {X 0,Y 439.343,Z 283.38,A -85,B 0,C 180,E1 -9222.208,E2 -9222.208} C_VEL
LIN {X 0,Y 439.36,Z 283.369,A -85,B 0,C 180,E1 -9225.266,E2 -9225.266} C_VEL
LIN {X 0,Y 439.365,Z 283.381,A -85,B 0,C 180,E1 -9228.743,E2 -9228.743} C_VEL
LIN {X 0,Y 439.356,Z 283.374,A -85,B 0,C 180,E1 -9231.607,E2 -9231.607} C_VEL
LIN {X 0,Y 439.379,Z 283.376,A -85,B 0,C 180,E1 -9234.843,E2 -9234.843} C_VEL
LIN {X 0,Y 439.354,Z 283.378,A -85,B 0,C 180,E1 -9238.138,E2 -9238.138} C_VEL
LIN {X 0,Y 439.415,Z 283.372,A -85,B 0,C 180,E1 -9241.597,E2 -9241.597} C_VEL
LIN {X 0,Y 439.38,Z 283.376,A -85,B 0,C 180,E1 -9244.414,E2 -9244.414} C_VEL
LIN {X 0,Y 439.345,Z 283.382,A -85,B 0,C 180,E1 -9247.424,E2 -9247.424} C_VEL
LIN {X 0,Y 439.424,Z 283.372,A -85,B 0,C 180,E1 -9250.662,E2 -9250.662} C_VEL
LIN {X 0,Y 439.444,Z 283.366,A -85,B 0,C 180,E1 -9254.224,E2 -9254.224} C_VEL
LIN {X 0,Y 439.491,Z 283.363,A -85,B 0,C 180,E1 -9258.001,E2 -9258.001} C_VEL
LIN {X 0,Y 439.53,Z 283.357,A -85,B 0,C 180,E1 -9261.726,E2 -9261.726} C_VEL
LIN {X 0,Y 439.597,Z 283.353,A -85,B 0,C 180,E1 -9264.495,E2 -9264.495} C_VEL
LIN {X 0,Y 439.617,Z 283.347,A -85,B 0,C 180,E1 -9268.167,E2 -9268.167} C_VEL
LIN {X 0,Y 439.745,Z 283.34,A -85,B 0,C 180,E1 -9270,E2 -9270} C_VEL
LIN {X 0,Y 439.62,Z 283.356,A -85,B 0,C 180,E1 -9270.936,E2 -9270.936} C_VEL
LIN {X 0,Y 439.193,Z 283.831,A -85,B 0,C 180,E1 -9271.356,E2 -9271.356} C_VEL
LIN {X 0,Y 437.752,Z 285.628,A -85,B 0,C 180,E1 -9271.889,E2 -9271.889} C_VEL
LIN {X 0,Y 435.022,Z 290.304,A -85,B 0,C 180,E1 -9272.717,E2 -9272.717} C_VEL
LIN {X 0,Y 434.499,Z 292.78,A -85,B 0,C 180,E1 -9273.147,E2 -9273.147} C_VEL
LIN {X 0,Y 434.583,Z 293.544,A -85,B 0,C 180,E1 -9273.297,E2 -9273.297} C_VEL
LIN {X 0,Y 435.258,Z 296.576,A -85,B 0,C 180,E1 -9273.876,E2 -9273.876} C_VEL
LIN {X 0,Y 441.089,Z 310.801,A -85,B 0,C 180,E1 -9274.497,E2 -9274.497} C_VEL
LIN {X 0,Y 443.474,Z 321.253,A -85,B 0,C 180,E1 -9274.829,E2 -9274.829} C_VEL
LIN {X 0,Y 441.186,Z 460.995,A -85,B 0,C 180,E1 -9277.206,E2 -9277.206} C_VEL
LIN {X 0,Y 440.654,Z 476.721,A -85,B 0,C 180,E1 -9277.655,E2 -9277.655} C_VEL
LIN {X 0,Y 439.906,Z 491.534,A -85,B 0,C 180,E1 -9278.266,E2 -9278.266} C_VEL
LIN {X 0,Y 438.972,Z 506.597,A -85,B 0,C 180,E1 -9279.096,E2 -9279.096} C_VEL
LIN {X 0,Y 437.959,Z 520.25,A -85,B 0,C 180,E1 -9280.05,E2 -9280.05} C_VEL
LIN {X 0,Y 436.84,Z 534.078,A -85,B 0,C 180,E1 -9281.248,E2 -9281.248} C_VEL
LIN {X 0,Y 435.711,Z 546.637,A -85,B 0,C 180,E1 -9282.577,E2 -9282.577} C_VEL
LIN {X 0,Y 434.657,Z 558.147,A -85,B 0,C 180,E1 -9284.046,E2 -9284.046} C_VEL
LIN {X 0,Y 433.756,Z 567.748,A -85,B 0,C 180,E1 -9285.506,E2 -9285.506} C_VEL
LIN {X 0,Y 432.941,Z 577.181,A -85,B 0,C 180,E1 -9287.232,E2 -9287.232} C_VEL
LIN {X 0,Y 432.358,Z 585.001,A -85,B 0,C 180,E1 -9288.971,E2 -9288.971} C_VEL
LIN {X 0,Y 431.914,Z 590.577,A -85,B 0,C 180,E1 -9290.477,E2 -9290.477} C_VEL
LIN {X 0,Y 431.634,Z 595.276,A -85,B 0,C 180,E1 -9291.992,E2 -9291.992} C_VEL
LIN {X 0,Y 431.384,Z 600.162,A -85,B 0,C 180,E1 -9294.034,E2 -9294.034} C_VEL
LIN {X 0,Y 431.118,Z 603.613,A -85,B 0,C 180,E1 -9296.112,E2 -9296.112} C_VEL
LIN {X 0,Y 431.029,Z 605.623,A -85,B 0,C 180,E1 -9298.218,E2 -9298.218} C_VEL
LIN {X 0,Y 431.018,Z 606.178,A -85,B 0,C 180,E1 -9300.362,E2 -9300.362} C_VEL
LIN {X 0,Y 431.033,Z 605.6,A -85,B 0,C 180,E1 -9302.025,E2 -9302.025} C_VEL
LIN {X 0,Y 431.092,Z 603.994,A -85,B 0,C 180,E1 -9303.757,E2 -9303.757} C_VEL
LIN {X 0,Y 431.338,Z 600.616,A -85,B 0,C 180,E1 -9305.912,E2 -9305.912} C_VEL
LIN {X 0,Y 431.573,Z 596.734,A -85,B 0,C 180,E1 -9307.637,E2 -9307.637} C_VEL
LIN {X 0,Y 431.881,Z 591.654,A -85,B 0,C 180,E1 -9309.392,E2 -9309.392} C_VEL
LIN {X 0,Y 432.342,Z 585.466,A -85,B 0,C 180,E1 -9311.105,E2 -9311.105} C_VEL
LIN {X 0,Y 433.036,Z 577.13,A -85,B 0,C 180,E1 -9312.971,E2 -9312.971} C_VEL
LIN {X 0,Y 433.866,Z 567.744,A -85,B 0,C 180,E1 -9314.688,E2 -9314.688} C_VEL
LIN {X 0,Y 434.843,Z 557.483,A -85,B 0,C 180,E1 -9316.246,E2 -9316.246} C_VEL
LIN {X 0,Y 435.953,Z 545.992,A -85,B 0,C 180,E1 -9317.696,E2 -9317.696} C_VEL
LIN {X 0,Y 437.032,Z 533.891,A -85,B 0,C 180,E1 -9318.969,E2 -9318.969} C_VEL
LIN {X 0,Y 438.232,Z 520.184,A -85,B 0,C 180,E1 -9320.149,E2 -9320.149} C_VEL
LIN {X 0,Y 439.22,Z 506.9,A -85,B 0,C 180,E1 -9321.08,E2 -9321.08} C_VEL
LIN {X 0,Y 440.123,Z 493.04,A -85,B 0,C 180,E1 -9321.852,E2 -9321.852} C_VEL
LIN {X 0,Y 440.925,Z 477.479,A -85,B 0,C 180,E1 -9322.509,E2 -9322.509} C_VEL
LIN {X 0,Y 441.524,Z 461.388,A -85,B 0,C 180,E1 -9322.972,E2 -9322.972} C_VEL
LIN {X 0,Y 443.888,Z 321.434,A -85,B 0,C 180,E1 -9325.379,E2 -9325.379} C_VEL
LIN {X 0,Y 441.146,Z 310.249,A -85,B 0,C 180,E1 -9325.762,E2 -9325.762} C_VEL
LIN {X 0,Y 435.441,Z 296.996,A -85,B 0,C 180,E1 -9326.409,E2 -9326.409} C_VEL
LIN {X 0,Y 432.312,Z 284.264,A -85,B 0,C 180,E1 -9329.148,E2 -9329.148} C_VEL
LIN {X 0,Y 432.368,Z 284.254,A -85,B 0,C 180,E1 -9331.878,E2 -9331.878} C_VEL
LIN {X 0,Y 432.336,Z 284.256,A -85,B 0,C 180,E1 -9335,E2 -9335} C_VEL
LIN {X 0,Y 432.342,Z 284.255,A -85,B 0,C 180,E1 -9338.047,E2 -9338.047} C_VEL
LIN {X 0,Y 432.371,Z 284.25,A -85,B 0,C 180,E1 -9341.031,E2 -9341.031} C_VEL
LIN {X 0,Y 432.416,Z 284.247,A -85,B 0,C 180,E1 -9343.962,E2 -9343.962} C_VEL
LIN {X 0,Y 432.445,Z 284.242,A -85,B 0,C 180,E1 -9347.805,E2 -9347.805} C_VEL
LIN {X 0,Y 432.479,Z 284.238,A -85,B 0,C 180,E1 -9351.592,E2 -9351.592} C_VEL
LIN {X 0,Y 432.579,Z 284.222,A -85,B 0,C 180,E1 -9354.408,E2 -9354.408} C_VEL
LIN {X 0,Y 432.592,Z 284.223,A -85,B 0,C 180,E1 -9358.14,E2 -9358.14} C_VEL
LIN {X 0,Y 432.72,Z 284.205,A -85,B 0,C 180,E1 -9360.002,E2 -9360.002} C_VEL
LIN {X 0,Y 432.577,Z 284.226,A -85,B 0,C 180,E1 -9362.795,E2 -9362.795} C_VEL
LIN {X 0,Y 432.576,Z 284.224,A -85,B 0,C 180,E1 -9365.596,E2 -9365.596} C_VEL
LIN {X 0,Y 432.453,Z 284.238,A -85,B 0,C 180,E1 -9368.412,E2 -9368.412} C_VEL
LIN {X 0,Y 432.449,Z 284.24,A -85,B 0,C 180,E1 -9372.198,E2 -9372.198} C_VEL
LIN {X 0,Y 432.421,Z 284.244,A -85,B 0,C 180,E1 -9376.041,E2 -9376.041} C_VEL
LIN {X 0,Y 432.378,Z 284.247,A -85,B 0,C 180,E1 -9379.486,E2 -9379.486} C_VEL
LIN {X 0,Y 432.302,Z 284.257,A -85,B 0,C 180,E1 -9382.966,E2 -9382.966} C_VEL
LIN {X 0,Y 432.309,Z 284.258,A -85,B 0,C 180,E1 -9386.037,E2 -9386.037} C_VEL
LIN {X 0,Y 432.32,Z 284.253,A -85,B 0,C 180,E1 -9389.19,E2 -9389.19} C_VEL
LIN {X 0,Y 432.314,Z 284.259,A -85,B 0,C 180,E1 -9392.445,E2 -9392.445} C_VEL
LIN {X 0,Y 432.326,Z 284.256,A -85,B 0,C 180,E1 -9395.82,E2 -9395.82} C_VEL
LIN {X 0,Y 432.294,Z 284.256,A -85,B 0,C 180,E1 -9399.35,E2 -9399.35} C_VEL
LIN {X 0,Y 432.298,Z 284.259,A -85,B 0,C 180,E1 -9401.802,E2 -9401.802} C_VEL
LIN {X 0,Y 432.328,Z 284.26,A -85,B 0,C 180,E1 -9404.349,E2 -9404.349} C_VEL
LIN {X 0,Y 432.298,Z 284.259,A -85,B 0,C 180,E1 -9407.02,E2 -9407.02} C_VEL
LIN {X 0,Y 432.285,Z 284.265,A -85,B 0,C 180,E1 -9409.829,E2 -9409.829} C_VEL
LIN {X 0,Y 432.294,Z 284.255,A -85,B 0,C 180,E1 -9413.022,E2 -9413.022} C_VEL
LIN {X 0,Y 432.356,Z 284.253,A -85,B 0,C 180,E1 -9415.998,E2 -9415.998} C_VEL
LIN {X 0,Y 432.361,Z 284.452,A -85,B 0,C 180,E1 -9417.656,E2 -9417.656} C_VEL
LIN {X 0,Y 435.767,Z 297.598,A -85,B 0,C 180,E1 -9420.232,E2 -9420.232} C_VEL
LIN {X 0,Y 438.201,Z 308.677,A -85,B 0,C 180,E1 -9422.284,E2 -9422.284} C_VEL
LIN {X 0,Y 437.555,Z 317.896,A -85,B 0,C 180,E1 -9423.773,E2 -9423.773} C_VEL
LIN {X 0,Y 442.738,Z 343.868,A -85,B 0,C 180,E1 -9424.597,E2 -9424.597} C_VEL
LIN {X 0,Y 443.608,Z 349.79,A -85,B 0,C 180,E1 -9424.759,E2 -9424.759} C_VEL
LIN {X 0,Y 441.26,Z 484.389,A -85,B 0,C 180,E1 -9427.064,E2 -9427.064} C_VEL
LIN {X 0,Y 440.598,Z 500.149,A -85,B 0,C 180,E1 -9427.512,E2 -9427.512} C_VEL
LIN {X 0,Y 439.814,Z 514.379,A -85,B 0,C 180,E1 -9428.096,E2 -9428.096} C_VEL
LIN {X 0,Y 438.75,Z 528.903,A -85,B 0,C 180,E1 -9428.875,E2 -9428.875} C_VEL
LIN {X 0,Y 437.737,Z 542.502,A -85,B 0,C 180,E1 -9429.808,E2 -9429.808} C_VEL
LIN {X 0,Y 436.461,Z 556.336,A -85,B 0,C 180,E1 -9430.97,E2 -9430.97} C_VEL
LIN {X 0,Y 435.43,Z 568.567,A -85,B 0,C 180,E1 -9432.23,E2 -9432.23} C_VEL
LIN {X 0,Y 434.427,Z 579.373,A -85,B 0,C 180,E1 -9433.555,E2 -9433.555} C_VEL
LIN {X 0,Y 433.529,Z 589.129,A -85,B 0,C 180,E1 -9434.968,E2 -9434.968} C_VEL
LIN {X 0,Y 432.703,Z 598.713,A -85,B 0,C 180,E1 -9436.618,E2 -9436.618} C_VEL
LIN {X 0,Y 432.167,Z 606.704,A -85,B 0,C 180,E1 -9438.272,E2 -9438.272} C_VEL
LIN {X 0,Y 431.645,Z 614.165,A -85,B 0,C 180,E1 -9440.157,E2 -9440.157} C_VEL
LIN {X 0,Y 431.408,Z 620.092,A -85,B 0,C 180,E1 -9442.041,E2 -9442.041} C_VEL
LIN {X 0,Y 431.2,Z 624.491,A -85,B 0,C 180,E1 -9443.841,E2 -9443.841} C_VEL
LIN {X 0,Y 431.209,Z 627.182,A -85,B 0,C 180,E1 -9445.326,E2 -9445.326} C_VEL
LIN {X 0,Y 431.22,Z 629.529,A -85,B 0,C 180,E1 -9447.198,E2 -9447.198} C_VEL
LIN {X 0,Y 431.168,Z 630.709,A -85,B 0,C 180,E1 -9449.066,E2 -9449.066} C_VEL
LIN {X 0,Y 431.168,Z 630.716,A -85,B 0,C 180,E1 -9450.934,E2 -9450.934} C_VEL
LIN {X 0,Y 431.22,Z 629.532,A -85,B 0,C 180,E1 -9452.803,E2 -9452.803} C_VEL
LIN {X 0,Y 431.212,Z 627.181,A -85,B 0,C 180,E1 -9454.675,E2 -9454.675} C_VEL
LIN {X 0,Y 431.282,Z 623.615,A -85,B 0,C 180,E1 -9456.55,E2 -9456.55} C_VEL
LIN {X 0,Y 431.455,Z 618.741,A -85,B 0,C 180,E1 -9458.43,E2 -9458.43} C_VEL
LIN {X 0,Y 431.74,Z 612.428,A -85,B 0,C 180,E1 -9460.315,E2 -9460.315} C_VEL
LIN {X 0,Y 432.215,Z 605.62,A -85,B 0,C 180,E1 -9461.965,E2 -9461.965} C_VEL
LIN {X 0,Y 432.815,Z 597.37,A -85,B 0,C 180,E1 -9463.618,E2 -9463.618} C_VEL
LIN {X 0,Y 433.618,Z 587.464,A -85,B 0,C 180,E1 -9465.271,E2 -9465.271} C_VEL
LIN {X 0,Y 434.587,Z 577.32,A -85,B 0,C 180,E1 -9466.681,E2 -9466.681} C_VEL
LIN {X 0,Y 435.621,Z 565.259,A -85,B 0,C 180,E1 -9468.093,E2 -9468.093} C_VEL
LIN {X 0,Y 436.684,Z 553.202,A -85,B 0,C 180,E1 -9469.264,E2 -9469.264} C_VEL
LIN {X 0,Y 437.801,Z 540.136,A -85,B 0,C 180,E1 -9470.313,E2 -9470.313} C_VEL
LIN {X 0,Y 438.801,Z 525.803,A -85,B 0,C 180,E1 -9471.246,E2 -9471.246} C_VEL
LIN {X 0,Y 439.803,Z 510.733,A -85,B 0,C 180,E1 -9472.003,E2 -9472.003} C_VEL
LIN {X 0,Y 440.529,Z 496.201,A -85,B 0,C 180,E1 -9472.543,E2 -9472.543} C_VEL
LIN {X 0,Y 441.056,Z 481.431,A -85,B 0,C 180,E1 -9472.917,E2 -9472.917} C_VEL
LIN {X 0,Y 443.223,Z 348.304,A -85,B 0,C 180,E1 -9475.171,E2 -9475.171} C_VEL
LIN {X 0,Y 437.446,Z 318.587,A -85,B 0,C 180,E1 -9476.058,E2 -9476.058} C_VEL
LIN {X 0,Y 438.052,Z 308.188,A -85,B 0,C 180,E1 -9477.727,E2 -9477.727} C_VEL
LIN {X 0,Y 435.197,Z 295.476,A -85,B 0,C 180,E1 -9480.041,E2 -9480.041} C_VEL
LIN {X 0,Y 432.321,Z 284.259,A -85,B 0,C 180,E1 -9482.207,E2 -9482.207} C_VEL
LIN {X 0,Y 432.342,Z 284.258,A -85,B 0,C 180,E1 -9485.63,E2 -9485.63} C_VEL
LIN {X 0,Y 432.32,Z 284.261,A -85,B 0,C 180,E1 -9488.71,E2 -9488.71} C_VEL
LIN {X 0,Y 432.303,Z 284.262,A -85,B 0,C 180,E1 -9491.8,E2 -9491.8} C_VEL
LIN {X 0,Y 432.332,Z 284.259,A -85,B 0,C 180,E1 -9494.347,E2 -9494.347} C_VEL
LIN {X 0,Y 432.303,Z 284.257,A -85,B 0,C 180,E1 -9497.017,E2 -9497.017} C_VEL
LIN {X 0,Y 432.288,Z 284.263,A -85,B 0,C 180,E1 -9499.827,E2 -9499.827} C_VEL
LIN {X 0,Y 432.294,Z 284.262,A -85,B 0,C 180,E1 -9503.02,E2 -9503.02} C_VEL
LIN {X 0,Y 432.331,Z 284.251,A -85,B 0,C 180,E1 -9506.001,E2 -9506.001} C_VEL
LIN {X 0,Y 432.342,Z 284.255,A -85,B 0,C 180,E1 -9509.489,E2 -9509.489} C_VEL
LIN {X 0,Y 432.325,Z 284.26,A -85,B 0,C 180,E1 -9511.872,E2 -9511.872} C_VEL
LIN {X 0,Y 432.346,Z 284.258,A -85,B 0,C 180,E1 -9515.546,E2 -9515.546} C_VEL
LIN {X 0,Y 432.346,Z 284.255,A -85,B 0,C 180,E1 -9519.045,E2 -9519.045} C_VEL
LIN {X 0,Y 432.354,Z 284.258,A -85,B 0,C 180,E1 -9522.009,E2 -9522.009} C_VEL
LIN {X 0,Y 432.384,Z 284.245,A -85,B 0,C 180,E1 -9524.925,E2 -9524.925} C_VEL
LIN {X 0,Y 432.448,Z 284.224,A -85,B 0,C 180,E1 -9527.802,E2 -9527.802} C_VEL
LIN {X 0,Y 432.44,Z 284.245,A -85,B 0,C 180,E1 -9531.588,E2 -9531.588} C_VEL
LIN {X 0,Y 432.544,Z 284.221,A -85,B 0,C 180,E1 -9534.404,E2 -9534.404} C_VEL
LIN {X 0,Y 432.583,Z 284.215,A -85,B 0,C 180,E1 -9538.136,E2 -9538.136} C_VEL
LIN {X 0,Y 432.592,Z 284.222,A -85,B 0,C 180,E1 -9539.998,E2 -9539.998} C_VEL
LIN {X 0,Y 432.557,Z 284.225,A -85,B 0,C 180,E1 -9542.792,E2 -9542.792} C_VEL
LIN {X 0,Y 432.475,Z 284.214,A -85,B 0,C 180,E1 -9546.449,E2 -9546.449} C_VEL
LIN {X 0,Y 432.412,Z 284.24,A -85,B 0,C 180,E1 -9549.352,E2 -9549.352} C_VEL
LIN {X 0,Y 432.421,Z 284.243,A -85,B 0,C 180,E1 -9552.801,E2 -9552.801} C_VEL
LIN {X 0,Y 432.384,Z 284.228,A -85,B 0,C 180,E1 -9556.468,E2 -9556.468} C_VEL
LIN {X 0,Y 432.326,Z 284.252,A -85,B 0,C 180,E1 -9559.959,E2 -9559.959} C_VEL
LIN {X 0,Y 432.298,Z 284.261,A -85,B 0,C 180,E1 -9562.963,E2 -9562.963} C_VEL
LIN {X 0,Y 432.304,Z 284.241,A -85,B 0,C 180,E1 -9566.034,E2 -9566.034} C_VEL
LIN {X 0,Y 432.31,Z 284.25,A -85,B 0,C 180,E1 -9569.188,E2 -9569.188} C_VEL
LIN {X 0,Y 432.307,Z 284.257,A -85,B 0,C 180,E1 -9572.442,E2 -9572.442} C_VEL
LIN {X 0,Y 432.321,Z 284.24,A -85,B 0,C 180,E1 -9575.817,E2 -9575.817} C_VEL
LIN {X 0,Y 432.287,Z 284.262,A -85,B 0,C 180,E1 -9579.347,E2 -9579.347} C_VEL
LIN {X 0,Y 432.293,Z 284.259,A -85,B 0,C 180,E1 -9581.799,E2 -9581.799} C_VEL
LIN {X 0,Y 432.316,Z 284.249,A -85,B 0,C 180,E1 -9584.346,E2 -9584.346} C_VEL
LIN {X 0,Y 432.3,Z 284.255,A -85,B 0,C 180,E1 -9587.015,E2 -9587.015} C_VEL
LIN {X 0,Y 432.315,Z 284.257,A -85,B 0,C 180,E1 -9589.82,E2 -9589.82} C_VEL
LIN {X 0,Y 432.289,Z 284.253,A -85,B 0,C 180,E1 -9593.021,E2 -9593.021} C_VEL
LIN {X 0,Y 432.341,Z 284.253,A -85,B 0,C 180,E1 -9595.996,E2 -9595.996} C_VEL
LIN {X 0,Y 432.329,Z 284.246,A -85,B 0,C 180,E1 -9599.489,E2 -9599.489} C_VEL
LIN {X 0,Y 432.373,Z 284.253,A -85,B 0,C 180,E1 -9602.927,E2 -9602.927} C_VEL
LIN {X 0,Y 432.349,Z 284.249,A -85,B 0,C 180,E1 -9606.022,E2 -9606.022} C_VEL
LIN {X 0,Y 432.332,Z 284.252,A -85,B 0,C 180,E1 -9609.045,E2 -9609.045} C_VEL
LIN {X 0,Y 432.359,Z 284.253,A -85,B 0,C 180,E1 -9612.01,E2 -9612.01} C_VEL
LIN {X 0,Y 432.377,Z 284.253,A -85,B 0,C 180,E1 -9614.926,E2 -9614.926} C_VEL
LIN {X 0,Y 432.463,Z 284.238,A -85,B 0,C 180,E1 -9617.803,E2 -9617.803} C_VEL
LIN {X 0,Y 432.474,Z 284.236,A -85,B 0,C 180,E1 -9621.59,E2 -9621.59} C_VEL
LIN {X 0,Y 432.574,Z 284.227,A -85,B 0,C 180,E1 -9624.406,E2 -9624.406} C_VEL
LIN {X 0,Y 432.586,Z 284.223,A -85,B 0,C 180,E1 -9628.138,E2 -9628.138} C_VEL
LIN {X 0,Y 432.715,Z 284.216,A -85,B 0,C 180,E1 -9630,E2 -9630} C_VEL
LIN {X 0,Y 432.579,Z 284.319,A -85,B 0,C 180,E1 -9631.396,E2 -9631.396} C_VEL
LIN {X 0,Y 434.583,Z 293.544,A -85,B 0,C 180,E1 -9633.297,E2 -9633.297} C_VEL
LIN {X 0,Y 435.272,Z 296.134,A -85,B 0,C 180,E1 -9633.665,E2 -9633.665} C_VEL
LIN {X 0,Y 436.42,Z 300.278,A -85,B 0,C 180,E1 -9633.976,E2 -9633.976} C_VEL
LIN {X 0,Y 437.409,Z 304.975,A -85,B 0,C 180,E1 -9634.165,E2 -9634.165} C_VEL
LIN {X 0,Y 437.761,Z 311.153,A -85,B 0,C 180,E1 -9634.3,E2 -9634.3} C_VEL
LIN {X 0,Y 437.018,Z 323.914,A -85,B 0,C 180,E1 -9634.488,E2 -9634.488} C_VEL
LIN {X 0,Y 434.61,Z 462.061,A -85,B 0,C 180,E1 -9636.878,E2 -9636.878} C_VEL
LIN {X 0,Y 433.98,Z 478.096,A -85,B 0,C 180,E1 -9637.356,E2 -9637.356} C_VEL
LIN {X 0,Y 433.276,Z 492.039,A -85,B 0,C 180,E1 -9637.948,E2 -9637.948} C_VEL
LIN {X 0,Y 432.326,Z 506.661,A -85,B 0,C 180,E1 -9638.766,E2 -9638.766} C_VEL
LIN {X 0,Y 431.242,Z 520.362,A -85,B 0,C 180,E1 -9639.734,E2 -9639.734} C_VEL
LIN {X 0,Y 430.095,Z 533.601,A -85,B 0,C 180,E1 -9640.888,E2 -9640.888} C_VEL
LIN {X 0,Y 428.993,Z 545.749,A -85,B 0,C 180,E1 -9642.176,E2 -9642.176} C_VEL
LIN {X 0,Y 427.837,Z 557.822,A -85,B 0,C 180,E1 -9643.721,E2 -9643.721} C_VEL
LIN {X 0,Y 426.835,Z 567.913,A -85,B 0,C 180,E1 -9645.274,E2 -9645.274} C_VEL
LIN {X 0,Y 426.003,Z 576.721,A -85,B 0,C 180,E1 -9646.9,E2 -9646.9} C_VEL
LIN {X 0,Y 425.331,Z 585.185,A -85,B 0,C 180,E1 -9648.796,E2 -9648.796} C_VEL
LIN {X 0,Y 424.719,Z 592.463,A -85,B 0,C 180,E1 -9650.84,E2 -9650.84} C_VEL
LIN {X 0,Y 424.421,Z 598.097,A -85,B 0,C 180,E1 -9652.9,E2 -9652.9} C_VEL
LIN {X 0,Y 424.196,Z 601.346,A -85,B 0,C 180,E1 -9654.468,E2 -9654.468} C_VEL
LIN {X 0,Y 423.982,Z 604.442,A -85,B 0,C 180,E1 -9656.586,E2 -9656.586} C_VEL
LIN {X 0,Y 423.887,Z 606.104,A -85,B 0,C 180,E1 -9658.738,E2 -9658.738} C_VEL
LIN {X 0,Y 423.917,Z 606.37,A -85,B 0,C 180,E1 -9660.453,E2 -9660.453} C_VEL
LIN {X 0,Y 423.97,Z 605.664,A -85,B 0,C 180,E1 -9662.289,E2 -9662.289} C_VEL
LIN {X 0,Y 424.04,Z 603.648,A -85,B 0,C 180,E1 -9664.298,E2 -9664.298} C_VEL
LIN {X 0,Y 424.239,Z 601.345,A -85,B 0,C 180,E1 -9665.738,E2 -9665.738} C_VEL
LIN {X 0,Y 424.519,Z 596.941,A -85,B 0,C 180,E1 -9667.772,E2 -9667.772} C_VEL
LIN {X 0,Y 424.956,Z 590.863,A -85,B 0,C 180,E1 -9669.854,E2 -9669.854} C_VEL
LIN {X 0,Y 425.497,Z 584.065,A -85,B 0,C 180,E1 -9671.685,E2 -9671.685} C_VEL
LIN {X 0,Y 426.213,Z 575.82,A -85,B 0,C 180,E1 -9673.49,E2 -9673.49} C_VEL
LIN {X 0,Y 427.044,Z 567.293,A -85,B 0,C 180,E1 -9675.043,E2 -9675.043} C_VEL
LIN {X 0,Y 428.038,Z 557.027,A -85,B 0,C 180,E1 -9676.61,E2 -9676.61} C_VEL
LIN {X 0,Y 429.265,Z 545.285,A -85,B 0,C 180,E1 -9678.094,E2 -9678.094} C_VEL
LIN {X 0,Y 430.365,Z 533.796,A -85,B 0,C 180,E1 -9679.312,E2 -9679.312} C_VEL
LIN {X 0,Y 431.583,Z 520.418,A -85,B 0,C 180,E1 -9680.48,E2 -9680.48} C_VEL
LIN {X 0,Y 432.676,Z 506.591,A -85,B 0,C 180,E1 -9681.459,E2 -9681.459} C_VEL
LIN {X 0,Y 433.669,Z 491.716,A -85,B 0,C 180,E1 -9682.284,E2 -9682.284} C_VEL
LIN {X 0,Y 434.457,Z 476.544,A -85,B 0,C 180,E1 -9682.914,E2 -9682.914} C_VEL
LIN {X 0,Y 435.024,Z 462.056,A -85,B 0,C 180,E1 -9683.334,E2 -9683.334} C_VEL
LIN {X 0,Y 437.563,Z 322.942,A -85,B 0,C 180,E1 -9685.763,E2 -9685.763} C_VEL
LIN {X 0,Y 435.189,Z 313.063,A -85,B 0,C 180,E1 -9686.109,E2 -9686.109} C_VEL
LIN {X 0,Y 428.318,Z 297.29,A -85,B 0,C 180,E1 -9686.898,E2 -9686.898} C_VEL
LIN {X 0,Y 425.336,Z 285.13,A -85,B 0,C 180,E1 -9689.586,E2 -9689.586} C_VEL
LIN {X 0,Y 425.332,Z 285.128,A -85,B 0,C 180,E1 -9693.157,E2 -9693.157} C_VEL
LIN {X 0,Y 425.291,Z 285.137,A -85,B 0,C 180,E1 -9696.636,E2 -9696.636} C_VEL
LIN {X 0,Y 425.313,Z 285.131,A -85,B 0,C 180,E1 -9700.366,E2 -9700.366} C_VEL
LIN {X 0,Y 425.374,Z 285.126,A -85,B 0,C 180,E1 -9703.69,E2 -9703.69} C_VEL
LIN {X 0,Y 425.398,Z 285.121,A -85,B 0,C 180,E1 -9707.6,E2 -9707.6} C_VEL
LIN {X 0,Y 425.429,Z 285.116,A -85,B 0,C 180,E1 -9711.451,E2 -9711.451} C_VEL
LIN {X 0,Y 425.536,Z 285.099,A -85,B 0,C 180,E1 -9714.315,E2 -9714.315} C_VEL
LIN {X 0,Y 425.561,Z 285.098,A -85,B 0,C 180,E1 -9718.109,E2 -9718.109} C_VEL
LIN {X 0,Y 425.69,Z 285.081,A -85,B 0,C 180,E1 -9720.002,E2 -9720.002} C_VEL
LIN {X 0,Y 425.53,Z 285.104,A -85,B 0,C 180,E1 -9722.842,E2 -9722.842} C_VEL
LIN {X 0,Y 425.532,Z 285.101,A -85,B 0,C 180,E1 -9725.688,E2 -9725.688} C_VEL
LIN {X 0,Y 425.398,Z 285.118,A -85,B 0,C 180,E1 -9728.552,E2 -9728.552} C_VEL
LIN {X 0,Y 425.402,Z 285.12,A -85,B 0,C 180,E1 -9732.403,E2 -9732.403} C_VEL
LIN {X 0,Y 425.379,Z 285.124,A -85,B 0,C 180,E1 -9736.313,E2 -9736.313} C_VEL
LIN {X 0,Y 425.32,Z 285.126,A -85,B 0,C 180,E1 -9739.637,E2 -9739.637} C_VEL
LIN {X 0,Y 425.279,Z 285.137,A -85,B 0,C 180,E1 -9742.34,E2 -9742.34} C_VEL
LIN {X 0,Y 425.249,Z 285.135,A -85,B 0,C 180,E1 -9745.449,E2 -9745.449} C_VEL
LIN {X 0,Y 425.301,Z 285.129,A -85,B 0,C 180,E1 -9748.862,E2 -9748.862} C_VEL
LIN {X 0,Y 425.254,Z 285.134,A -85,B 0,C 180,E1 -9751.929,E2 -9751.929} C_VEL
LIN {X 0,Y 425.286,Z 285.131,A -85,B 0,C 180,E1 -9755.338,E2 -9755.338} C_VEL
LIN {X 0,Y 425.27,Z 285.131,A -85,B 0,C 180,E1 -9758.903,E2 -9758.903} C_VEL
LIN {X 0,Y 425.252,Z 285.138,A -85,B 0,C 180,E1 -9762.657,E2 -9762.657} C_VEL
LIN {X 0,Y 425.28,Z 285.134,A -85,B 0,C 180,E1 -9765.285,E2 -9765.285} C_VEL
LIN {X 0,Y 425.244,Z 285.14,A -85,B 0,C 180,E1 -9768.619,E2 -9768.619} C_VEL
LIN {X 0,Y 425.273,Z 285.136,A -85,B 0,C 180,E1 -9771.1,E2 -9771.1} C_VEL
LIN {X 0,Y 425.293,Z 285.134,A -85,B 0,C 180,E1 -9774.665,E2 -9774.665} C_VEL
LIN {X 0,Y 425.286,Z 285.262,A -85,B 0,C 180,E1 -9777.204,E2 -9777.204} C_VEL
LIN {X 0,Y 428.846,Z 298.847,A -85,B 0,C 180,E1 -9779.934,E2 -9779.934} C_VEL
LIN {X 0,Y 431.419,Z 310.561,A -85,B 0,C 180,E1 -9782.145,E2 -9782.145} C_VEL
LIN {X 0,Y 430.91,Z 317.927,A -85,B 0,C 180,E1 -9783.328,E2 -9783.328} C_VEL
LIN {X 0,Y 436.171,Z 343.97,A -85,B 0,C 180,E1 -9784.177,E2 -9784.177} C_VEL
LIN {X 0,Y 437.225,Z 350.312,A -85,B 0,C 180,E1 -9784.364,E2 -9784.364} C_VEL
LIN {X 0,Y 434.757,Z 484.604,A -85,B 0,C 180,E1 -9786.701,E2 -9786.701} C_VEL
LIN {X 0,Y 434.041,Z 500.233,A -85,B 0,C 180,E1 -9787.155,E2 -9787.155} C_VEL
LIN {X 0,Y 433.149,Z 515.333,A -85,B 0,C 180,E1 -9787.791,E2 -9787.791} C_VEL
LIN {X 0,Y 432.109,Z 528.83,A -85,B 0,C 180,E1 -9788.535,E2 -9788.535} C_VEL
LIN {X 0,Y 431.046,Z 542.383,A -85,B 0,C 180,E1 -9789.48,E2 -9789.48} C_VEL
LIN {X 0,Y 429.698,Z 556.184,A -85,B 0,C 180,E1 -9790.659,E2 -9790.659} C_VEL
LIN {X 0,Y 428.554,Z 569.143,A -85,B 0,C 180,E1 -9792.021,E2 -9792.021} C_VEL
LIN {X 0,Y 427.359,Z 580.984,A -85,B 0,C 180,E1 -9793.521,E2 -9793.521} C_VEL
LIN {X 0,Y 426.35,Z 591.909,A -85,B 0,C 180,E1 -9795.197,E2 -9795.197} C_VEL
LIN {X 0,Y 425.474,Z 601.391,A -85,B 0,C 180,E1 -9796.955,E2 -9796.955} C_VEL
LIN {X 0,Y 425.069,Z 608.564,A -85,B 0,C 180,E1 -9798.557,E2 -9798.557} C_VEL
LIN {X 0,Y 424.514,Z 615.614,A -85,B 0,C 180,E1 -9800.471,E2 -9800.471} C_VEL
LIN {X 0,Y 424.285,Z 621.163,A -85,B 0,C 180,E1 -9802.386,E2 -9802.386} C_VEL
LIN {X 0,Y 424.107,Z 625.36,A -85,B 0,C 180,E1 -9804.294,E2 -9804.294} C_VEL
LIN {X 0,Y 424.056,Z 628.304,A -85,B 0,C 180,E1 -9806.199,E2 -9806.199} C_VEL
LIN {X 0,Y 424.126,Z 630.062,A -85,B 0,C 180,E1 -9808.101,E2 -9808.101} C_VEL
LIN {X 0,Y 424.083,Z 630.665,A -85,B 0,C 180,E1 -9810,E2 -9810} C_VEL
LIN {X 0,Y 424.126,Z 630.063,A -85,B 0,C 180,E1 -9811.9,E2 -9811.9} C_VEL
LIN {X 0,Y 424.056,Z 628.292,A -85,B 0,C 180,E1 -9813.801,E2 -9813.801} C_VEL
LIN {X 0,Y 424.128,Z 625.336,A -85,B 0,C 180,E1 -9815.706,E2 -9815.706} C_VEL
LIN {X 0,Y 424.276,Z 621.122,A -85,B 0,C 180,E1 -9817.615,E2 -9817.615} C_VEL
LIN {X 0,Y 424.523,Z 615.536,A -85,B 0,C 180,E1 -9819.529,E2 -9819.529} C_VEL
LIN {X 0,Y 425.068,Z 608.432,A -85,B 0,C 180,E1 -9821.444,E2 -9821.444} C_VEL
LIN {X 0,Y 425.471,Z 601.252,A -85,B 0,C 180,E1 -9823.042,E2 -9823.042} C_VEL
LIN {X 0,Y 426.305,Z 591.668,A -85,B 0,C 180,E1 -9824.805,E2 -9824.805} C_VEL
LIN {X 0,Y 427.345,Z 580.603,A -85,B 0,C 180,E1 -9826.48,E2 -9826.48} C_VEL
LIN {X 0,Y 428.384,Z 569.289,A -85,B 0,C 180,E1 -9827.909,E2 -9827.909} C_VEL
LIN {X 0,Y 429.527,Z 556.738,A -85,B 0,C 180,E1 -9829.226,E2 -9829.226} C_VEL
LIN {X 0,Y 430.704,Z 544.452,A -85,B 0,C 180,E1 -9830.288,E2 -9830.288} C_VEL
LIN {X 0,Y 431.766,Z 531.179,A -85,B 0,C 180,E1 -9831.233,E2 -9831.233} C_VEL
LIN {X 0,Y 432.796,Z 516.863,A -85,B 0,C 180,E1 -9832.045,E2 -9832.045} C_VEL
LIN {X 0,Y 433.616,Z 501.79,A -85,B 0,C 180,E1 -9832.697,E2 -9832.697} C_VEL
LIN {X 0,Y 434.344,Z 487.201,A -85,B 0,C 180,E1 -9833.134,E2 -9833.134} C_VEL
LIN {X 0,Y 434.838,Z 463.471,A -85,B 0,C 180,E1 -9833.579,E2 -9833.579} C_VEL
LIN {X 0,Y 436.695,Z 349.001,A -85,B 0,C 180,E1 -9835.544,E2 -9835.544} C_VEL
LIN {X 0,Y 430.701,Z 318.308,A -85,B 0,C 180,E1 -9836.498,E2 -9836.498} C_VEL
LIN {X 0,Y 431.236,Z 310.009,A -85,B 0,C 180,E1 -9837.851,E2 -9837.851} C_VEL
LIN {X 0,Y 428.205,Z 296.592,A -85,B 0,C 180,E1 -9840.337,E2 -9840.337} C_VEL
LIN {X 0,Y 425.27,Z 285.137,A -85,B 0,C 180,E1 -9842.587,E2 -9842.587} C_VEL
LIN {X 0,Y 425.28,Z 285.137,A -85,B 0,C 180,E1 -9845.927,E2 -9845.927} C_VEL
LIN {X 0,Y 425.259,Z 285.139,A -85,B 0,C 180,E1 -9849.036,E2 -9849.036} C_VEL
LIN {X 0,Y 425.257,Z 285.134,A -85,B 0,C 180,E1 -9852.655,E2 -9852.655} C_VEL
LIN {X 0,Y 425.284,Z 285.134,A -85,B 0,C 180,E1 -9855.282,E2 -9855.282} C_VEL
LIN {X 0,Y 425.248,Z 285.142,A -85,B 0,C 180,E1 -9858.617,E2 -9858.617} C_VEL
LIN {X 0,Y 425.275,Z 285.13,A -85,B 0,C 180,E1 -9861.098,E2 -9861.098} C_VEL
LIN {X 0,Y 425.291,Z 285.128,A -85,B 0,C 180,E1 -9864.662,E2 -9864.662} C_VEL
LIN {X 0,Y 425.262,Z 285.14,A -85,B 0,C 180,E1 -9868.072,E2 -9868.072} C_VEL
LIN {X 0,Y 425.303,Z 285.132,A -85,B 0,C 180,E1 -9871.365,E2 -9871.365} C_VEL
LIN {X 0,Y 425.256,Z 285.138,A -85,B 0,C 180,E1 -9874.551,E2 -9874.551} C_VEL
LIN {X 0,Y 425.289,Z 285.138,A -85,B 0,C 180,E1 -9877.729,E2 -9877.729} C_VEL
LIN {X 0,Y 425.358,Z 285.121,A -85,B 0,C 180,E1 -9880.703,E2 -9880.703} C_VEL
LIN {X 0,Y 425.382,Z 285.125,A -85,B 0,C 180,E1 -9883.687,E2 -9883.687} C_VEL
LIN {X 0,Y 425.404,Z 285.1,A -85,B 0,C 180,E1 -9887.597,E2 -9887.597} C_VEL
LIN {X 0,Y 425.388,Z 285.121,A -85,B 0,C 180,E1 -9891.447,E2 -9891.447} C_VEL
LIN {X 0,Y 425.502,Z 285.099,A -85,B 0,C 180,E1 -9894.311,E2 -9894.311} C_VEL
LIN {X 0,Y 425.552,Z 285.091,A -85,B 0,C 180,E1 -9898.106,E2 -9898.106} C_VEL
LIN {X 0,Y 425.427,Z 285.114,A -85,B 0,C 180,E1 -9900.945,E2 -9900.945} C_VEL
LIN {X 0,Y 425.512,Z 285.103,A -85,B 0,C 180,E1 -9902.839,E2 -9902.839} C_VEL
LIN {X 0,Y 425.437,Z 285.089,A -85,B 0,C 180,E1 -9906.447,E2 -9906.447} C_VEL
LIN {X 0,Y 425.373,Z 285.119,A -85,B 0,C 180,E1 -9909.508,E2 -9909.508} C_VEL
LIN {X 0,Y 425.384,Z 285.12,A -85,B 0,C 180,E1 -9912.901,E2 -9912.901} C_VEL
LIN {X 0,Y 425.336,Z 285.106,A -85,B 0,C 180,E1 -9916.596,E2 -9916.596} C_VEL
LIN {X 0,Y 425.317,Z 285.127,A -85,B 0,C 180,E1 -9919.634,E2 -9919.634} C_VEL
LIN {X 0,Y 425.276,Z 285.132,A -85,B 0,C 180,E1 -9922.337,E2 -9922.337} C_VEL
LIN {X 0,Y 425.246,Z 285.125,A -85,B 0,C 180,E1 -9925.446,E2 -9925.446} C_VEL
LIN {X 0,Y 425.287,Z 285.12,A -85,B 0,C 180,E1 -9928.857,E2 -9928.857} C_VEL
LIN {X 0,Y 425.248,Z 285.136,A -85,B 0,C 180,E1 -9931.926,E2 -9931.926} C_VEL
LIN {X 0,Y 425.28,Z 285.121,A -85,B 0,C 180,E1 -9935.335,E2 -9935.335} C_VEL
LIN {X 0,Y 425.266,Z 285.129,A -85,B 0,C 180,E1 -9938.899,E2 -9938.899} C_VEL
LIN {X 0,Y 425.245,Z 285.139,A -85,B 0,C 180,E1 -9942.654,E2 -9942.654} C_VEL
LIN {X 0,Y 425.268,Z 285.123,A -85,B 0,C 180,E1 -9945.282,E2 -9945.282} C_VEL
LIN {X 0,Y 425.251,Z 285.138,A -85,B 0,C 180,E1 -9948.619,E2 -9948.619} C_VEL
LIN {X 0,Y 425.281,Z 285.132,A -85,B 0,C 180,E1 -9951.1,E2 -9951.1} C_VEL
LIN {X 0,Y 425.281,Z 285.13,A -85,B 0,C 180,E1 -9954.663,E2 -9954.663} C_VEL
LIN {X 0,Y 425.247,Z 285.135,A -85,B 0,C 180,E1 -9958.072,E2 -9958.072} C_VEL
LIN {X 0,Y 425.313,Z 285.13,A -85,B 0,C 180,E1 -9961.367,E2 -9961.367} C_VEL
LIN {X 0,Y 425.336,Z 285.123,A -85,B 0,C 180,E1 -9963.504,E2 -9963.504} C_VEL
LIN {X 0,Y 425.266,Z 285.137,A -85,B 0,C 180,E1 -9966.633,E2 -9966.633} C_VEL
LIN {X 0,Y 425.277,Z 285.128,A -85,B 0,C 180,E1 -9969.694,E2 -9969.694} C_VEL
LIN {X 0,Y 425.323,Z 285.129,A -85,B 0,C 180,E1 -9972.697,E2 -9972.697} C_VEL
LIN {X 0,Y 425.335,Z 285.126,A -85,B 0,C 180,E1 -9975.65,E2 -9975.65} C_VEL
LIN {X 0,Y 425.353,Z 285.129,A -85,B 0,C 180,E1 -9978.564,E2 -9978.564} C_VEL
LIN {X 0,Y 425.52,Z 285.104,A -85,B 0,C 180,E1 -9982.407,E2 -9982.407} C_VEL
LIN {X 0,Y 425.531,Z 285.104,A -85,B 0,C 180,E1 -9984.313,E2 -9984.313} C_VEL
LIN {X 0,Y 425.555,Z 285.098,A -85,B 0,C 180,E1 -9988.107,E2 -9988.107} C_VEL
LIN {X 0,Y 425.685,Z 285.092,A -85,B 0,C 180,E1 -9990,E2 -9990} C_VEL
LIN {X 0,Y 425.568,Z 285.199,A -85,B 0,C 180,E1 -9991.035,E2 -9991.035} C_VEL
LIN {X 0,Y 428.092,Z 296.766,A -85,B 0,C 180,E1 -9993.421,E2 -9993.421} C_VEL
LIN {X 0,Y 434.967,Z 313.418,A -85,B 0,C 180,E1 -9994.169,E2 -9994.169} C_VEL
LIN {X 0,Y 437.043,Z 322.658,A -85,B 0,C 180,E1 -9994.467,E2 -9994.467} C_VEL
LIN {X 0,Y 437.018,Z 323.914,A -85,B 0,C 180,E1 -9994.488,E2 -9994.488} C_VEL
LIN {X 0,Y 436.289,Z 329.764,A -85,B 0,C 180,E1 -9994.551,E2 -9994.551} C_VEL
LIN {X 0,Y 430.669,Z 348.804,A -85,B 0,C 180,E1 -9994.557,E2 -9994.557} C_VEL
LIN {X 0,Y 430.008,Z 354.65,A -85,B 0,C 180,E1 -9994.626,E2 -9994.626} C_VEL
LIN {X 0,Y 428.084,Z 461.822,A -85,B 0,C 180,E1 -9996.51,E2 -9996.51} C_VEL
LIN {X 0,Y 427.482,Z 477.204,A -85,B 0,C 180,E1 -9996.964,E2 -9996.964} C_VEL
LIN {X 0,Y 426.611,Z 492.849,A -85,B 0,C 180,E1 -9997.635,E2 -9997.635} C_VEL
LIN {X 0,Y 425.616,Z 507.501,A -85,B 0,C 180,E1 -9998.476,E2 -9998.476} C_VEL
LIN {X 0,Y 424.555,Z 520.459,A -85,B 0,C 180,E1 -9999.408,E2 -9999.408} C_VEL
LIN {X 0,Y 423.389,Z 533.1,A -85,B 0,C 180,E1 -10000.52,E2 -10000.52} C_VEL
LIN {X 0,Y 422.194,Z 545.888,A -85,B 0,C 180,E1 -10001.887,E2 -10001.887} C_VEL
LIN {X 0,Y 421.127,Z 556.592,A -85,B 0,C 180,E1 -10003.265,E2 -10003.265} C_VEL
LIN {X 0,Y 420.092,Z 566.526,A -85,B 0,C 180,E1 -10004.78,E2 -10004.78} C_VEL
LIN {X 0,Y 419.235,Z 574.963,A -85,B 0,C 180,E1 -10006.307,E2 -10006.307} C_VEL
LIN {X 0,Y 418.445,Z 583.249,A -85,B 0,C 180,E1 -10008.102,E2 -10008.102} C_VEL
LIN {X 0,Y 417.981,Z 589.344,A -85,B 0,C 180,E1 -10009.687,E2 -10009.687} C_VEL
LIN {X 0,Y 417.501,Z 595.657,A -85,B 0,C 180,E1 -10011.735,E2 -10011.735} C_VEL
LIN {X 0,Y 417.223,Z 600.548,A -85,B 0,C 180,E1 -10013.845,E2 -10013.845} C_VEL
LIN {X 0,Y 416.937,Z 604.006,A -85,B 0,C 180,E1 -10015.992,E2 -10015.992} C_VEL
LIN {X 0,Y 416.802,Z 606.027,A -85,B 0,C 180,E1 -10018.171,E2 -10018.171} C_VEL
LIN {X 0,Y 416.818,Z 606.586,A -85,B 0,C 180,E1 -10020.385,E2 -10020.385} C_VEL
LIN {X 0,Y 416.882,Z 605.692,A -85,B 0,C 180,E1 -10022.554,E2 -10022.554} C_VEL
LIN {X 0,Y 416.952,Z 603.924,A -85,B 0,C 180,E1 -10024.322,E2 -10024.322} C_VEL
LIN {X 0,Y 417.285,Z 599.878,A -85,B 0,C 180,E1 -10026.718,E2 -10026.718} C_VEL
LIN {X 0,Y 417.562,Z 595.619,A -85,B 0,C 180,E1 -10028.516,E2 -10028.516} C_VEL
LIN {X 0,Y 417.993,Z 590.208,A -85,B 0,C 180,E1 -10030.291,E2 -10030.291} C_VEL
LIN {X 0,Y 418.623,Z 583.062,A -85,B 0,C 180,E1 -10032.184,E2 -10032.184} C_VEL
LIN {X 0,Y 419.377,Z 575.147,A -85,B 0,C 180,E1 -10033.899,E2 -10033.899} C_VEL
LIN {X 0,Y 420.392,Z 565.625,A -85,B 0,C 180,E1 -10035.611,E2 -10035.611} C_VEL
LIN {X 0,Y 421.444,Z 555.025,A -85,B 0,C 180,E1 -10037.199,E2 -10037.199} C_VEL
LIN {X 0,Y 422.704,Z 543.666,A -85,B 0,C 180,E1 -10038.611,E2 -10038.611} C_VEL
LIN {X 0,Y 423.899,Z 531.444,A -85,B 0,C 180,E1 -10039.88,E2 -10039.88} C_VEL
LIN {X 0,Y 425.134,Z 518.561,A -85,B 0,C 180,E1 -10040.982,E2 -10040.982} C_VEL
LIN {X 0,Y 426.263,Z 504.885,A -85,B 0,C 180,E1 -10041.931,E2 -10041.931} C_VEL
LIN {X 0,Y 427.196,Z 490.826,A -85,B 0,C 180,E1 -10042.704,E2 -10042.704} C_VEL
LIN {X 0,Y 428.038,Z 475.882,A -85,B 0,C 180,E1 -10043.319,E2 -10043.319} C_VEL
LIN {X 0,Y 428.614,Z 460.642,A -85,B 0,C 180,E1 -10043.751,E2 -10043.751} C_VEL
LIN {X 0,Y 431.214,Z 324.129,A -85,B 0,C 180,E1 -10046.171,E2 -10046.171} C_VEL
LIN {X 0,Y 429.17,Z 315.805,A -85,B 0,C 180,E1 -10046.473,E2 -10046.473} C_VEL
LIN {X 0,Y 421.125,Z 297.452,A -85,B 0,C 180,E1 -10047.441,E2 -10047.441} C_VEL
LIN {X 0,Y 418.269,Z 286.01,A -85,B 0,C 180,E1 -10050.045,E2 -10050.045} C_VEL
LIN {X 0,Y 418.288,Z 286.005,A -85,B 0,C 180,E1 -10053.024,E2 -10053.024} C_VEL
LIN {X 0,Y 418.272,Z 286.011,A -85,B 0,C 180,E1 -10056.22,E2 -10056.22} C_VEL
LIN {X 0,Y 418.235,Z 286.02,A -85,B 0,C 180,E1 -10059.338,E2 -10059.338} C_VEL
LIN {X 0,Y 418.273,Z 286.009,A -85,B 0,C 180,E1 -10062.398,E2 -10062.398} C_VEL
LIN {X 0,Y 418.288,Z 286.008,A -85,B 0,C 180,E1 -10065.404,E2 -10065.404} C_VEL
LIN {X 0,Y 418.301,Z 286.004,A -85,B 0,C 180,E1 -10068.37,E2 -10068.37} C_VEL
LIN {X 0,Y 418.501,Z 285.977,A -85,B 0,C 180,E1 -10072.281,E2 -10072.281} C_VEL
LIN {X 0,Y 418.496,Z 285.975,A -85,B 0,C 180,E1 -10074.219,E2 -10074.219} C_VEL
LIN {X 0,Y 418.531,Z 285.974,A -85,B 0,C 180,E1 -10078.077,E2 -10078.077} C_VEL
LIN {X 0,Y 418.66,Z 285.957,A -85,B 0,C 180,E1 -10080.002,E2 -10080.002} C_VEL
LIN {X 0,Y 418.485,Z 285.982,A -85,B 0,C 180,E1 -10082.889,E2 -10082.889} C_VEL
LIN {X 0,Y 418.49,Z 285.978,A -85,B 0,C 180,E1 -10085.785,E2 -10085.785} C_VEL
LIN {X 0,Y 418.367,Z 285.995,A -85,B 0,C 180,E1 -10088.697,E2 -10088.697} C_VEL
LIN {X 0,Y 418.304,Z 286.001,A -85,B 0,C 180,E1 -10091.633,E2 -10091.633} C_VEL
LIN {X 0,Y 418.293,Z 286.004,A -85,B 0,C 180,E1 -10094.599,E2 -10094.599} C_VEL
LIN {X 0,Y 418.271,Z 286.004,A -85,B 0,C 180,E1 -10097.606,E2 -10097.606} C_VEL
LIN {X 0,Y 418.242,Z 286.011,A -85,B 0,C 180,E1 -10100.665,E2 -10100.665} C_VEL
LIN {X 0,Y 418.247,Z 286.007,A -85,B 0,C 180,E1 -10103.785,E2 -10103.785} C_VEL
LIN {X 0,Y 418.207,Z 286.015,A -85,B 0,C 180,E1 -10107.046,E2 -10107.046} C_VEL
LIN {X 0,Y 418.233,Z 286.014,A -85,B 0,C 180,E1 -10110.274,E2 -10110.274} C_VEL
LIN {X 0,Y 418.226,Z 286.011,A -85,B 0,C 180,E1 -10113.68,E2 -10113.68} C_VEL
LIN {X 0,Y 418.227,Z 286.01,A -85,B 0,C 180,E1 -10117.227,E2 -10117.227} C_VEL
LIN {X 0,Y 418.202,Z 286.014,A -85,B 0,C 180,E1 -10120.868,E2 -10120.868} C_VEL
LIN {X 0,Y 418.198,Z 286.016,A -85,B 0,C 180,E1 -10123.729,E2 -10123.729} C_VEL
LIN {X 0,Y 418.195,Z 286.02,A -85,B 0,C 180,E1 -10126.449,E2 -10126.449} C_VEL
LIN {X 0,Y 418.204,Z 286.016,A -85,B 0,C 180,E1 -10129.134,E2 -10129.134} C_VEL
LIN {X 0,Y 418.231,Z 286.007,A -85,B 0,C 180,E1 -10132.776,E2 -10132.776} C_VEL
LIN {X 0,Y 418.246,Z 286.014,A -85,B 0,C 180,E1 -10136.324,E2 -10136.324} C_VEL
LIN {X 0,Y 418.246,Z 286.062,A -85,B 0,C 180,E1 -10136.73,E2 -10136.73} C_VEL
LIN {X 0,Y 422.115,Z 300.802,A -85,B 0,C 180,E1 -10139.76,E2 -10139.76} C_VEL
LIN {X 0,Y 424.578,Z 312.035,A -85,B 0,C 180,E1 -10141.925,E2 -10141.925} C_VEL
LIN {X 0,Y 424.256,Z 317.479,A -85,B 0,C 180,E1 -10142.845,E2 -10142.845} C_VEL
LIN {X 0,Y 429.397,Z 342.689,A -85,B 0,C 180,E1 -10143.697,E2 -10143.697} C_VEL
LIN {X 0,Y 430.878,Z 351.503,A -85,B 0,C 180,E1 -10143.966,E2 -10143.966} C_VEL
LIN {X 0,Y 428.253,Z 484.781,A -85,B 0,C 180,E1 -10146.326,E2 -10146.326} C_VEL
LIN {X 0,Y 427.502,Z 500.362,A -85,B 0,C 180,E1 -10146.789,E2 -10146.789} C_VEL
LIN {X 0,Y 426.676,Z 514.278,A -85,B 0,C 180,E1 -10147.381,E2 -10147.381} C_VEL
LIN {X 0,Y 425.504,Z 528.776,A -85,B 0,C 180,E1 -10148.185,E2 -10148.185} C_VEL
LIN {X 0,Y 424.361,Z 542.296,A -85,B 0,C 180,E1 -10149.142,E2 -10149.142} C_VEL
LIN {X 0,Y 422.976,Z 556.076,A -85,B 0,C 180,E1 -10150.339,E2 -10150.339} C_VEL
LIN {X 0,Y 421.818,Z 568.613,A -85,B 0,C 180,E1 -10151.677,E2 -10151.677} C_VEL
LIN {X 0,Y 420.516,Z 580.823,A -85,B 0,C 180,E1 -10153.245,E2 -10153.245} C_VEL
LIN {X 0,Y 419.396,Z 591.728,A -85,B 0,C 180,E1 -10154.946,E2 -10154.946} C_VEL
LIN {X 0,Y 418.476,Z 601.495,A -85,B 0,C 180,E1 -10156.795,E2 -10156.795} C_VEL
LIN {X 0,Y 418.04,Z 608.381,A -85,B 0,C 180,E1 -10158.362,E2 -10158.362} C_VEL
LIN {X 0,Y 417.438,Z 615.428,A -85,B 0,C 180,E1 -10160.308,E2 -10160.308} C_VEL
LIN {X 0,Y 417.198,Z 620.975,A -85,B 0,C 180,E1 -10162.255,E2 -10162.255} C_VEL
LIN {X 0,Y 417.009,Z 625.168,A -85,B 0,C 180,E1 -10164.197,E2 -10164.197} C_VEL
LIN {X 0,Y 416.97,Z 628.109,A -85,B 0,C 180,E1 -10166.135,E2 -10166.135} C_VEL
LIN {X 0,Y 417.053,Z 629.863,A -85,B 0,C 180,E1 -10168.069,E2 -10168.069} C_VEL
LIN {X 0,Y 417.003,Z 630.461,A -85,B 0,C 180,E1 -10170,E2 -10170} C_VEL
LIN {X 0,Y 417.053,Z 629.856,A -85,B 0,C 180,E1 -10171.932,E2 -10171.932} C_VEL
LIN {X 0,Y 416.971,Z 628.076,A -85,B 0,C 180,E1 -10173.866,E2 -10173.866} C_VEL
LIN {X 0,Y 417.048,Z 625.112,A -85,B 0,C 180,E1 -10175.803,E2 -10175.803} C_VEL
LIN {X 0,Y 417.193,Z 620.887,A -85,B 0,C 180,E1 -10177.745,E2 -10177.745} C_VEL
LIN {X 0,Y 417.446,Z 615.289,A -85,B 0,C 180,E1 -10179.692,E2 -10179.692} C_VEL
